//     Term 1 (APS4322-7000)/APS Outputs/Current D 1X0 <-> Data Pointer/DCurrentSetPoints[6]
//     Term 1 (APS4322-7000)/APS Outputs/Current D 1X1 <-> Data Pointer/DCurrentSetPoints[7]
//     Term 1 (APS4322-7000)/APS Outputs/Current D 1X2 <-> Data Pointer/DCurrentSetPoints[8]
//     Term 1 (APS4322-7000)/APS Outputs/Current D 2X0 <-> Data Pointer/DCurrentSetPoints[12]
//     Term 1 (APS4322-7000)/APS Outputs/Current D 2X1 <-> Data Pointer/DCurrentSetPoints[13]
//     Term 1 (APS4322-7000)/APS Outputs/Current D 2X2 <-> Data Pointer/DCurrentSetPoints[14]
//     Term 1 (APS4322-7000)/APS Outputs/Current D 3X0 <-> Data Pointer/DCurrentSetPoints[18]
//     Term 1 (APS4322-7000)/APS Outputs/Current D 3X1 <-> Data Pointer/DCurrentSetPoints[19]
//     Term 1 (APS4322-7000)/APS Outputs/Current D 3X2 <-> Data Pointer/DCurrentSetPoints[20]
//     Term 1 (APS4322-7000)/APS Outputs/Current D 0Y0 <-> Data Pointer/DCurrentSetPoints[3]
//     Term 1 (APS4322-7000)/APS Outputs/Current D 0Y1 <-> Data Pointer/DCurrentSetPoints[4]
//     Term 1 (APS4322-7000)/APS Outputs/Current D 0Y2 <-> Data Pointer/DCurrentSetPoints[5]
//     Term 1 (APS4322-7000)/APS Outputs/Current D 1Y0 <-> Data Pointer/DCurrentSetPoints[9]
//     Term 1 (APS4322-7000)/APS Outputs/Current D 1Y1 <-> Data Pointer/DCurrentSetPoints[10]
//     Term 1 (APS4322-7000)/APS Outputs/Current D 1Y2 <-> Data Pointer/DCurrentSetPoints[11]
//     Term 1 (APS4322-7000)/APS Outputs/Current D 2Y0 <-> Data Pointer/DCurrentSetPoints[15]
//     Term 1 (APS4322-7000)/APS Outputs/Current D 2Y1 <-> Data Pointer/DCurrentSetPoints[16]
//     Term 1 (APS4322-7000)/APS Outputs/Current D 2Y2 <-> Data Pointer/DCurrentSetPoints[17]
//     Term 1 (APS4322-7000)/APS Outputs/Current D 3Y0 <-> Data Pointer/DCurrentSetPoints[21]
//     Term 1 (APS4322-7000)/APS Outputs/Current D 3Y1 <-> Data Pointer/DCurrentSetPoints[22]
//     Term 1 (APS4322-7000)/APS Outputs/Current D 3Y2 <-> Data Pointer/DCurrentSetPoints[23]
//     Term 1 (APS4322-7000)/APS Outputs/Current Q 0X0 <-> Data Pointer/QCurrentSetPoints[0]
//     Term 1 (APS4322-7000)/APS Outputs/Current Q 0X1 <-> Data Pointer/QCurrentSetPoints[1]
//     Term 1 (APS4322-7000)/APS Outputs/Current Q 0X2 <-> Data Pointer/QCurrentSetPoints[2]
//     Term 1 (APS4322-7000)/APS Outputs/Current Q 1X0 <-> Data Pointer/QCurrentSetPoints[6]
//     Term 1 (APS4322-7000)/APS Outputs/Current Q 1X1 <-> Data Pointer/QCurrentSetPoints[7]
//     Term 1 (APS4322-7000)/APS Outputs/Current Q 1X2 <-> Data Pointer/QCurrentSetPoints[8]
//     Term 1 (APS4322-7000)/APS Outputs/Current Q 2X0 <-> Data Pointer/QCurrentSetPoints[12]
//     Term 1 (APS4322-7000)/APS Outputs/Current Q 2X1 <-> Data Pointer/QCurrentSetPoints[13]
//     Term 1 (APS4322-7000)/APS Outputs/Current Q 2X2 <-> Data Pointer/QCurrentSetPoints[14]
//     Term 1 (APS4322-7000)/APS Outputs/Current Q 3X0 <-> Data Pointer/QCurrentSetPoints[18]
//     Term 1 (APS4322-7000)/APS Outputs/Current Q 3X1 <-> Data Pointer/QCurrentSetPoints[19]
//     Term 1 (APS4322-7000)/APS Outputs/Current Q 3X2 <-> Data Pointer/QCurrentSetPoints[20]
//     Term 1 (APS4322-7000)/APS Outputs/Current Q 0Y0 <-> Data Pointer/QCurrentSetPoints[3]
//     Term 1 (APS4322-7000)/APS Outputs/Current Q 0Y1 <-> Data Pointer/QCurrentSetPoints[4]
//     Term 1 (APS4322-7000)/APS Outputs/Current Q 0Y2 <-> Data Pointer/QCurrentSetPoints[5]
//     Term 1 (APS4322-7000)/APS Outputs/Current Q 1Y0 <-> Data Pointer/QCurrentSetPoints[9]
//     Term 1 (APS4322-7000)/APS Outputs/Current Q 1Y1 <-> Data Pointer/QCurrentSetPoints[10]
//     Term 1 (APS4322-7000)/APS Outputs/Current Q 1Y2 <-> Data Pointer/QCurrentSetPoints[11]
//     Term 1 (APS4322-7000)/APS Outputs/Current Q 2Y0 <-> Data Pointer/QCurrentSetPoints[15]
//     Term 1 (APS4322-7000)/APS Outputs/Current Q 2Y1 <-> Data Pointer/QCurrentSetPoints[16]
//     Term 1 (APS4322-7000)/APS Outputs/Current Q 2Y2 <-> Data Pointer/QCurrentSetPoints[17]
//     Term 1 (APS4322-7000)/APS Outputs/Current Q 3Y0 <-> Data Pointer/QCurrentSetPoints[21]
//     Term 1 (APS4322-7000)/APS Outputs/Current Q 3Y1 <-> Data Pointer/QCurrentSetPoints[22]
//     Term 1 (APS4322-7000)/APS Outputs/Current Q 3Y2 <-> Data Pointer/QCurrentSetPoints[23]
//     Term 1 (APS4322-7000)/APS Outputs/PhiE 0X0 <-> Data Pointer/PhiSetPoints[0]
//     Term 1 (APS4322-7000)/APS Outputs/PhiE 0X1 <-> Data Pointer/PhiSetPoints[1]
//     Term 1 (APS4322-7000)/APS Outputs/PhiE 0X2 <-> Data Pointer/PhiSetPoints[2]
//     Term 1 (APS4322-7000)/APS Outputs/PhiE 1X0 <-> Data Pointer/PhiSetPoints[6]
//     Term 1 (APS4322-7000)/APS Outputs/PhiE 1X1 <-> Data Pointer/PhiSetPoints[7]
//     Term 1 (APS4322-7000)/APS Outputs/PhiE 1X2 <-> Data Pointer/PhiSetPoints[8]
//     Term 1 (APS4322-7000)/APS Outputs/PhiE 2X0 <-> Data Pointer/PhiSetPoints[12]
//     Term 1 (APS4322-7000)/APS Outputs/PhiE 2X1 <-> Data Pointer/PhiSetPoints[13]
//     Term 1 (APS4322-7000)/APS Outputs/PhiE 2X2 <-> Data Pointer/PhiSetPoints[14]
//     Term 1 (APS4322-7000)/APS Outputs/PhiE 3X0 <-> Data Pointer/PhiSetPoints[18]
//     Term 1 (APS4322-7000)/APS Outputs/PhiE 3X1 <-> Data Pointer/PhiSetPoints[19]
//     Term 1 (APS4322-7000)/APS Outputs/PhiE 3X2 <-> Data Pointer/PhiSetPoints[20]
//     Term 1 (APS4322-7000)/APS Outputs/PhiE 0Y0 <-> Data Pointer/PhiSetPoints[3]
//     Term 1 (APS4322-7000)/APS Outputs/PhiE 0Y1 <-> Data Pointer/PhiSetPoints[4]
//     Term 1 (APS4322-7000)/APS Outputs/PhiE 0Y2 <-> Data Pointer/PhiSetPoints[5]
//     Term 1 (APS4322-7000)/APS Outputs/PhiE 1Y0 <-> Data Pointer/PhiSetPoints[9]
//     Term 1 (APS4322-7000)/APS Outputs/PhiE 1Y1 <-> Data Pointer/PhiSetPoints[10]
//     Term 1 (APS4322-7000)/APS Outputs/PhiE 1Y2 <-> Data Pointer/PhiSetPoints[11]
//     Term 1 (APS4322-7000)/APS Outputs/PhiE 2Y0 <-> Data Pointer/PhiSetPoints[15]
//     Term 1 (APS4322-7000)/APS Outputs/PhiE 2Y1 <-> Data Pointer/PhiSetPoints[16]
//     Term 1 (APS4322-7000)/APS Outputs/PhiE 2Y2 <-> Data Pointer/PhiSetPoints[17]
//     Term 1 (APS4322-7000)/APS Outputs/PhiE 3Y0 <-> Data Pointer/PhiSetPoints[21]
//     Term 1 (APS4322-7000)/APS Outputs/PhiE 3Y1 <-> Data Pointer/PhiSetPoints[22]
//     Term 1 (APS4322-7000)/APS Outputs/PhiE 3Y2 <-> Data Pointer/PhiSetPoints[23]
//     Term 1 (APS4322-7000)/Term 2 (APS4322-5000)/FB Inputs/A{0..8 step 2} X-Field <-> Data Pointer/HallSensorFieldsXYZ[{0..12 step 3}]  (5 links)
//     Term 1 (APS4322-7000)/Term 2 (APS4322-5000)/FB Inputs/A{0..8 step 2} Y-Field <-> Data Pointer/HallSensorFieldsXYZ[{1..13 step 3}]  (5 links)
//     Term 1 (APS4322-7000)/Term 2 (APS4322-5000)/FB Inputs/A{0..8 step 2} Z-Field <-> Data Pointer/HallSensorFieldsXYZ[{2..14 step 3}]  (5 links)
//     Term 1 (APS4322-7000)/Term 2 (APS4322-5000)/FB Inputs/B{1..9 step 2} X-Field <-> Data Pointer/HallSensorFieldsXYZ[{15..27 step 3}]  (5 links)
//     Term 1 (APS4322-7000)/Term 2 (APS4322-5000)/FB Inputs/B{1..9 step 2} Y-Field <-> Data Pointer/HallSensorFieldsXYZ[{16..28 step 3}]  (5 links)
//     Term 1 (APS4322-7000)/Term 2 (APS4322-5000)/FB Inputs/B{1..9 step 2} Z-Field <-> Data Pointer/HallSensorFieldsXYZ[{17..29 step 3}]  (5 links)
//     Term 1 (APS4322-7000)/Term 2 (APS4322-5000)/FB Inputs/C{0..8 step 2} X-Field <-> Data Pointer/HallSensorFieldsXYZ[{30..42 step 3}]  (5 links)
//     Term 1 (APS4322-7000)/Term 2 (APS4322-5000)/FB Inputs/C{0..8 step 2} Y-Field <-> Data Pointer/HallSensorFieldsXYZ[{31..43 step 3}]  (5 links)
//     Term 1 (APS4322-7000)/Term 2 (APS4322-5000)/FB Inputs/C{0..8 step 2} Z-Field <-> Data Pointer/HallSensorFieldsXYZ[{32..44 step 3}]  (5 links)
//     Term 1 (APS4322-7000)/Term 2 (APS4322-5000)/FB Inputs/D{1..9 step 2} X-Field <-> Data Pointer/HallSensorFieldsXYZ[{45..57 step 3}]  (5 links)
//     Term 1 (APS4322-7000)/Term 2 (APS4322-5000)/FB Inputs/D{1..9 step 2} Y-Field <-> Data Pointer/HallSensorFieldsXYZ[{46..58 step 3}]  (5 links)
//     Term 1 (APS4322-7000)/Term 2 (APS4322-5000)/FB Inputs/D{1..9 step 2} Z-Field <-> Data Pointer/HallSensorFieldsXYZ[{47..59 step 3}]  (5 links)
//     Term 1 (APS4322-7000)/Term 2 (APS4322-5000)/FB Inputs/E{0..8 step 2} X-Field <-> Data Pointer/HallSensorFieldsXYZ[{60..72 step 3}]  (5 links)
//     Term 1 (APS4322-7000)/Term 2 (APS4322-5000)/FB Inputs/E{0..8 step 2} Y-Field <-> Data Pointer/HallSensorFieldsXYZ[{61..73 step 3}]  (5 links)
//     Term 1 (APS4322-7000)/Term 2 (APS4322-5000)/FB Inputs/E{0..8 step 2} Z-Field <-> Data Pointer/HallSensorFieldsXYZ[{62..74 step 3}]  (5 links)
//     Term 1 (APS4322-7000)/Term 2 (APS4322-5000)/FB Inputs/F{1..9 step 2} X-Field <-> Data Pointer/HallSensorFieldsXYZ[{75..87 step 3}]  (5 links)
//     Term 1 (APS4322-7000)/Term 2 (APS4322-5000)/FB Inputs/F{1..9 step 2} Y-Field <-> Data Pointer/HallSensorFieldsXYZ[{76..88 step 3}]  (5 links)
//     Term 1 (APS4322-7000)/Term 2 (APS4322-5000)/FB Inputs/F{1..9 step 2} Z-Field <-> Data Pointer/HallSensorFieldsXYZ[{77..89 step 3}]  (5 links)
//     Term 1 (APS4322-7000)/Term 2 (APS4322-5000)/FB Inputs/G{0..8 step 2} X-Field <-> Data Pointer/HallSensorFieldsXYZ[{90..102 step 3}]  (5 links)
//     Term 1 (APS4322-7000)/Term 2 (APS4322-5000)/FB Inputs/G{0..8 step 2} Y-Field <-> Data Pointer/HallSensorFieldsXYZ[{91..103 step 3}]  (5 links)
//     Term 1 (APS4322-7000)/Term 2 (APS4322-5000)/FB Inputs/G{0..8 step 2} Z-Field <-> Data Pointer/HallSensorFieldsXYZ[{92..104 step 3}]  (5 links)
//     Term 1 (APS4322-7000)/Term 2 (APS4322-5000)/FB Inputs/H{1..9 step 2} X-Field <-> Data Pointer/HallSensorFieldsXYZ[{105..117 step 3}]  (5 links)
//     Term 1 (APS4322-7000)/Term 2 (APS4322-5000)/FB Inputs/H{1..9 step 2} Y-Field <-> Data Pointer/HallSensorFieldsXYZ[{106..118 step 3}]  (5 links)
//     Term 1 (APS4322-7000)/Term 2 (APS4322-5000)/FB Inputs/H{1..9 step 2} Z-Field <-> Data Pointer/HallSensorFieldsXYZ[{107..119 step 3}]  (5 links)
//     Term 1 (APS4322-7000)/Term 2 (APS4322-5000)/FB Inputs/I{0..8 step 2} X-Field <-> Data Pointer/HallSensorFieldsXYZ[{120..132 step 3}]  (5 links)
//     Term 1 (APS4322-7000)/Term 2 (APS4322-5000)/FB Inputs/I{0..8 step 2} Y-Field <-> Data Pointer/HallSensorFieldsXYZ[{121..133 step 3}]  (5 links)
//     Term 1 (APS4322-7000)/Term 2 (APS4322-5000)/FB Inputs/I{0..8 step 2} Z-Field <-> Data Pointer/HallSensorFieldsXYZ[{122..134 step 3}]  (5 links)
//     Term 1 (APS4322-7000)/Term 2 (APS4322-5000)/FB Inputs/J{1..9 step 2} X-Field <-> Data Pointer/HallSensorFieldsXYZ[{135..147 step 3}]  (5 links)
//     Term 1 (APS4322-7000)/Term 2 (APS4322-5000)/FB Inputs/J{1..9 step 2} Y-Field <-> Data Pointer/HallSensorFieldsXYZ[{136..148 step 3}]  (5 links)
//     Term 1 (APS4322-7000)/Term 2 (APS4322-5000)/FB Inputs/J{1..9 step 2} Z-Field <-> Data Pointer/HallSensorFieldsXYZ[{137..149 step 3}]  (5 links)
//     Term 1 (APS4322-7000)/Term 2 (APS4322-5000)/FB Inputs/Status <-> Data Pointer/FeedbackStatus
//   Device 6 (EtherCAT) <-> TcCOM Objects/XPlanar/Part1/APS4322_P1_4
//     Term 3 (APS4322-7000)/APS Comm Inputs/CommStatusWord <-> Data Pointer/MoverCommStatusWord
//     Term 3 (APS4322-7000)/APS Comm Inputs/Data {1..4} <-> Data Pointer/MoverCommDataIn[{0..3}]  (4 links)
//     Term 3 (APS4322-7000)/APS Comm Outputs/CommControlWord <-> Data Pointer/MoverCommControlWord
//     Term 3 (APS4322-7000)/APS Comm Outputs/Data 1 <-> Data Pointer/MoverCommDataOut
//     Term 3 (APS4322-7000)/APS Diagdata/DC Link Voltage <-> Data Pointer/DcLinkVoltage
//     Term 3 (APS4322-7000)/APS Diagdata/Power supply current <-> Data Pointer/PowerSupplyCurrent
//     Term 3 (APS4322-7000)/APS Inputs/StatusWord <-> Data Pointer/PowerUnitStatusWord
//     Term 3 (APS4322-7000)/APS Outputs/ControlWord <-> Data Pointer/PowerUnitControlWord
//     Term 3 (APS4322-7000)/APS Outputs/Current D 0X0 <-> Data Pointer/DCurrentSetPoints[0]
//     Term 3 (APS4322-7000)/APS Outputs/Current D 0X1 <-> Data Pointer/DCurrentSetPoints[1]
//     Term 3 (APS4322-7000)/APS Outputs/Current D 0X2 <-> Data Pointer/DCurrentSetPoints[2]
//     Term 3 (APS4322-7000)/APS Outputs/Current D 1X0 <-> Data Pointer/DCurrentSetPoints[6]
//     Term 3 (APS4322-7000)/APS Outputs/Current D 1X1 <-> Data Pointer/DCurrentSetPoints[7]
//     Term 3 (APS4322-7000)/APS Outputs/Current D 1X2 <-> Data Pointer/DCurrentSetPoints[8]
//     Term 3 (APS4322-7000)/APS Outputs/Current D 2X0 <-> Data Pointer/DCurrentSetPoints[12]
//     Term 3 (APS4322-7000)/APS Outputs/Current D 2X1 <-> Data Pointer/DCurrentSetPoints[13]
//     Term 3 (APS4322-7000)/APS Outputs/Current D 2X2 <-> Data Pointer/DCurrentSetPoints[14]
//     Term 3 (APS4322-7000)/APS Outputs/Current D 3X0 <-> Data Pointer/DCurrentSetPoints[18]
//     Term 3 (APS4322-7000)/APS Outputs/Current D 3X1 <-> Data Pointer/DCurrentSetPoints[19]
//     Term 3 (APS4322-7000)/APS Outputs/Current D 3X2 <-> Data Pointer/DCurrentSetPoints[20]
//     Term 3 (APS4322-7000)/APS Outputs/Current D 0Y0 <-> Data Pointer/DCurrentSetPoints[3]
//     Term 3 (APS4322-7000)/APS Outputs/Current D 0Y1 <-> Data Pointer/DCurrentSetPoints[4]
//     Term 3 (APS4322-7000)/APS Outputs/Current D 0Y2 <-> Data Pointer/DCurrentSetPoints[5]
//     Term 3 (APS4322-7000)/APS Outputs/Current D 1Y0 <-> Data Pointer/DCurrentSetPoints[9]
//     Term 3 (APS4322-7000)/APS Outputs/Current D 1Y1 <-> Data Pointer/DCurrentSetPoints[10]
//     Term 3 (APS4322-7000)/APS Outputs/Current D 1Y2 <-> Data Pointer/DCurrentSetPoints[11]
//     Term 3 (APS4322-7000)/APS Outputs/Current D 2Y0 <-> Data Pointer/DCurrentSetPoints[15]
//     Term 3 (APS4322-7000)/APS Outputs/Current D 2Y1 <-> Data Pointer/DCurrentSetPoints[16]
//     Term 3 (APS4322-7000)/APS Outputs/Current D 2Y2 <-> Data Pointer/DCurrentSetPoints[17]
//     Term 3 (APS4322-7000)/APS Outputs/Current D 3Y0 <-> Data Pointer/DCurrentSetPoints[21]
//     Term 3 (APS4322-7000)/APS Outputs/Current D 3Y1 <-> Data Pointer/DCurrentSetPoints[22]
//     Term 3 (APS4322-7000)/APS Outputs/Current D 3Y2 <-> Data Pointer/DCurrentSetPoints[23]
//     Term 3 (APS4322-7000)/APS Outputs/Current Q 0X0 <-> Data Pointer/QCurrentSetPoints[0]
//     Term 3 (APS4322-7000)/APS Outputs/Current Q 0X1 <-> Data Pointer/QCurrentSetPoints[1]
//     Term 3 (APS4322-7000)/APS Outputs/Current Q 0X2 <-> Data Pointer/QCurrentSetPoints[2]
//     Term 3 (APS4322-7000)/APS Outputs/Current Q 1X0 <-> Data Pointer/QCurrentSetPoints[6]
//     Term 3 (APS4322-7000)/APS Outputs/Current Q 1X1 <-> Data Pointer/QCurrentSetPoints[7]
//     Term 3 (APS4322-7000)/APS Outputs/Current Q 1X2 <-> Data Pointer/QCurrentSetPoints[8]
//     Term 3 (APS4322-7000)/APS Outputs/Current Q 2X0 <-> Data Pointer/QCurrentSetPoints[12]
//     Term 3 (APS4322-7000)/APS Outputs/Current Q 2X1 <-> Data Pointer/QCurrentSetPoints[13]
//     Term 3 (APS4322-7000)/APS Outputs/Current Q 2X2 <-> Data Pointer/QCurrentSetPoints[14]
//     Term 3 (APS4322-7000)/APS Outputs/Current Q 3X0 <-> Data Pointer/QCurrentSetPoints[18]
//     Term 3 (APS4322-7000)/APS Outputs/Current Q 3X1 <-> Data Pointer/QCurrentSetPoints[19]
//     Term 3 (APS4322-7000)/APS Outputs/Current Q 3X2 <-> Data Pointer/QCurrentSetPoints[20]
//     Term 3 (APS4322-7000)/APS Outputs/Current Q 0Y0 <-> Data Pointer/QCurrentSetPoints[3]
//     Term 3 (APS4322-7000)/APS Outputs/Current Q 0Y1 <-> Data Pointer/QCurrentSetPoints[4]
//     Term 3 (APS4322-7000)/APS Outputs/Current Q 0Y2 <-> Data Pointer/QCurrentSetPoints[5]
//     Term 3 (APS4322-7000)/APS Outputs/Current Q 1Y0 <-> Data Pointer/QCurrentSetPoints[9]
//     Term 3 (APS4322-7000)/APS Outputs/Current Q 1Y1 <-> Data Pointer/QCurrentSetPoints[10]
//     Term 3 (APS4322-7000)/APS Outputs/Current Q 1Y2 <-> Data Pointer/QCurrentSetPoints[11]
//     Term 3 (APS4322-7000)/APS Outputs/Current Q 2Y0 <-> Data Pointer/QCurrentSetPoints[15]
//     Term 3 (APS4322-7000)/APS Outputs/Current Q 2Y1 <-> Data Pointer/QCurrentSetPoints[16]
//     Term 3 (APS4322-7000)/APS Outputs/Current Q 2Y2 <-> Data Pointer/QCurrentSetPoints[17]
//     Term 3 (APS4322-7000)/APS Outputs/Current Q 3Y0 <-> Data Pointer/QCurrentSetPoints[21]
//     Term 3 (APS4322-7000)/APS Outputs/Current Q 3Y1 <-> Data Pointer/QCurrentSetPoints[22]
//     Term 3 (APS4322-7000)/APS Outputs/Current Q 3Y2 <-> Data Pointer/QCurrentSetPoints[23]
//     Term 3 (APS4322-7000)/APS Outputs/PhiE 0X0 <-> Data Pointer/PhiSetPoints[0]
//     Term 3 (APS4322-7000)/APS Outputs/PhiE 0X1 <-> Data Pointer/PhiSetPoints[1]
//     Term 3 (APS4322-7000)/APS Outputs/PhiE 0X2 <-> Data Pointer/PhiSetPoints[2]
//     Term 3 (APS4322-7000)/APS Outputs/PhiE 1X0 <-> Data Pointer/PhiSetPoints[6]
//     Term 3 (APS4322-7000)/APS Outputs/PhiE 1X1 <-> Data Pointer/PhiSetPoints[7]
//     Term 3 (APS4322-7000)/APS Outputs/PhiE 1X2 <-> Data Pointer/PhiSetPoints[8]
//     Term 3 (APS4322-7000)/APS Outputs/PhiE 2X0 <-> Data Pointer/PhiSetPoints[12]
//     Term 3 (APS4322-7000)/APS Outputs/PhiE 2X1 <-> Data Pointer/PhiSetPoints[13]
//     Term 3 (APS4322-7000)/APS Outputs/PhiE 2X2 <-> Data Pointer/PhiSetPoints[14]
//     Term 3 (APS4322-7000)/APS Outputs/PhiE 3X0 <-> Data Pointer/PhiSetPoints[18]
//     Term 3 (APS4322-7000)/APS Outputs/PhiE 3X1 <-> Data Pointer/PhiSetPoints[19]
//     Term 3 (APS4322-7000)/APS Outputs/PhiE 3X2 <-> Data Pointer/PhiSetPoints[20]
//     Term 3 (APS4322-7000)/APS Outputs/PhiE 0Y0 <-> Data Pointer/PhiSetPoints[3]
//     Term 3 (APS4322-7000)/APS Outputs/PhiE 0Y1 <-> Data Pointer/PhiSetPoints[4]
//     Term 3 (APS4322-7000)/APS Outputs/PhiE 0Y2 <-> Data Pointer/PhiSetPoints[5]
//     Term 3 (APS4322-7000)/APS Outputs/PhiE 1Y0 <-> Data Pointer/PhiSetPoints[9]
//     Term 3 (APS4322-7000)/APS Outputs/PhiE 1Y1 <-> Data Pointer/PhiSetPoints[10]
//     Term 3 (APS4322-7000)/APS Outputs/PhiE 1Y2 <-> Data Pointer/PhiSetPoints[11]
//     Term 3 (APS4322-7000)/APS Outputs/PhiE 2Y0 <-> Data Pointer/PhiSetPoints[15]
//     Term 3 (APS4322-7000)/APS Outputs/PhiE 2Y1 <-> Data Pointer/PhiSetPoints[16]
//     Term 3 (APS4322-7000)/APS Outputs/PhiE 2Y2 <-> Data Pointer/PhiSetPoints[17]
//     Term 3 (APS4322-7000)/APS Outputs/PhiE 3Y0 <-> Data Pointer/PhiSetPoints[21]
//     Term 3 (APS4322-7000)/APS Outputs/PhiE 3Y1 <-> Data Pointer/PhiSetPoints[22]
//     Term 3 (APS4322-7000)/APS Outputs/PhiE 3Y2 <-> Data Pointer/PhiSetPoints[23]
//     Term 3 (APS4322-7000)/Term 4 (APS4322-5000)/FB Inputs/A{0..8 step 2} X-Field <-> Data Pointer/HallSensorFieldsXYZ[{0..12 step 3}]  (5 links)
//     Term 3 (APS4322-7000)/Term 4 (APS4322-5000)/FB Inputs/A{0..8 step 2} Y-Field <-> Data Pointer/HallSensorFieldsXYZ[{1..13 step 3}]  (5 links)
//     Term 3 (APS4322-7000)/Term 4 (APS4322-5000)/FB Inputs/A{0..8 step 2} Z-Field <-> Data Pointer/HallSensorFieldsXYZ[{2..14 step 3}]  (5 links)
//     Term 3 (APS4322-7000)/Term 4 (APS4322-5000)/FB Inputs/B{1..9 step 2} X-Field <-> Data Pointer/HallSensorFieldsXYZ[{15..27 step 3}]  (5 links)
//     Term 3 (APS4322-7000)/Term 4 (APS4322-5000)/FB Inputs/B{1..9 step 2} Y-Field <-> Data Pointer/HallSensorFieldsXYZ[{16..28 step 3}]  (5 links)
//     Term 3 (APS4322-7000)/Term 4 (APS4322-5000)/FB Inputs/B{1..9 step 2} Z-Field <-> Data Pointer/HallSensorFieldsXYZ[{17..29 step 3}]  (5 links)
//     Term 3 (APS4322-7000)/Term 4 (APS4322-5000)/FB Inputs/C{0..8 step 2} X-Field <-> Data Pointer/HallSensorFieldsXYZ[{30..42 step 3}]  (5 links)
//     Term 3 (APS4322-7000)/Term 4 (APS4322-5000)/FB Inputs/C{0..8 step 2} Y-Field <-> Data Pointer/HallSensorFieldsXYZ[{31..43 step 3}]  (5 links)
//     Term 3 (APS4322-7000)/Term 4 (APS4322-5000)/FB Inputs/C{0..8 step 2} Z-Field <-> Data Pointer/HallSensorFieldsXYZ[{32..44 step 3}]  (5 links)
//     Term 3 (APS4322-7000)/Term 4 (APS4322-5000)/FB Inputs/D{1..9 step 2} X-Field <-> Data Pointer/HallSensorFieldsXYZ[{45..57 step 3}]  (5 links)
//     Term 3 (APS4322-7000)/Term 4 (APS4322-5000)/FB Inputs/D{1..9 step 2} Y-Field <-> Data Pointer/HallSensorFieldsXYZ[{46..58 step 3}]  (5 links)
//     Term 3 (APS4322-7000)/Term 4 (APS4322-5000)/FB Inputs/D{1..9 step 2} Z-Field <-> Data Pointer/HallSensorFieldsXYZ[{47..59 step 3}]  (5 links)
//     Term 3 (APS4322-7000)/Term 4 (APS4322-5000)/FB Inputs/E{0..8 step 2} X-Field <-> Data Pointer/HallSensorFieldsXYZ[{60..72 step 3}]  (5 links)
//     Term 3 (APS4322-7000)/Term 4 (APS4322-5000)/FB Inputs/E{0..8 step 2} Y-Field <-> Data Pointer/HallSensorFieldsXYZ[{61..73 step 3}]  (5 links)
//     Term 3 (APS4322-7000)/Term 4 (APS4322-5000)/FB Inputs/E{0..8 step 2} Z-Field <-> Data Pointer/HallSensorFieldsXYZ[{62..74 step 3}]  (5 links)
//     Term 3 (APS4322-7000)/Term 4 (APS4322-5000)/FB Inputs/F{1..9 step 2} X-Field <-> Data Pointer/HallSensorFieldsXYZ[{75..87 step 3}]  (5 links)
//     Term 3 (APS4322-7000)/Term 4 (APS4322-5000)/FB Inputs/F{1..9 step 2} Y-Field <-> Data Pointer/HallSensorFieldsXYZ[{76..88 step 3}]  (5 links)
//     Term 3 (APS4322-7000)/Term 4 (APS4322-5000)/FB Inputs/F{1..9 step 2} Z-Field <-> Data Pointer/HallSensorFieldsXYZ[{77..89 step 3}]  (5 links)
//     Term 3 (APS4322-7000)/Term 4 (APS4322-5000)/FB Inputs/G{0..8 step 2} X-Field <-> Data Pointer/HallSensorFieldsXYZ[{90..102 step 3}]  (5 links)
//     Term 3 (APS4322-7000)/Term 4 (APS4322-5000)/FB Inputs/G{0..8 step 2} Y-Field <-> Data Pointer/HallSensorFieldsXYZ[{91..103 step 3}]  (5 links)
//     Term 3 (APS4322-7000)/Term 4 (APS4322-5000)/FB Inputs/G{0..8 step 2} Z-Field <-> Data Pointer/HallSensorFieldsXYZ[{92..104 step 3}]  (5 links)
//     Term 3 (APS4322-7000)/Term 4 (APS4322-5000)/FB Inputs/H{1..9 step 2} X-Field <-> Data Pointer/HallSensorFieldsXYZ[{105..117 step 3}]  (5 links)
//     Term 3 (APS4322-7000)/Term 4 (APS4322-5000)/FB Inputs/H{1..9 step 2} Y-Field <-> Data Pointer/HallSensorFieldsXYZ[{106..118 step 3}]  (5 links)
//     Term 3 (APS4322-7000)/Term 4 (APS4322-5000)/FB Inputs/H{1..9 step 2} Z-Field <-> Data Pointer/HallSensorFieldsXYZ[{107..119 step 3}]  (5 links)
//     Term 3 (APS4322-7000)/Term 4 (APS4322-5000)/FB Inputs/I{0..8 step 2} X-Field <-> Data Pointer/HallSensorFieldsXYZ[{120..132 step 3}]  (5 links)
//     Term 3 (APS4322-7000)/Term 4 (APS4322-5000)/FB Inputs/I{0..8 step 2} Y-Field <-> Data Pointer/HallSensorFieldsXYZ[{121..133 step 3}]  (5 links)
//     Term 3 (APS4322-7000)/Term 4 (APS4322-5000)/FB Inputs/I{0..8 step 2} Z-Field <-> Data Pointer/HallSensorFieldsXYZ[{122..134 step 3}]  (5 links)
//     Term 3 (APS4322-7000)/Term 4 (APS4322-5000)/FB Inputs/J{1..9 step 2} X-Field <-> Data Pointer/HallSensorFieldsXYZ[{135..147 step 3}]  (5 links)
//     Term 3 (APS4322-7000)/Term 4 (APS4322-5000)/FB Inputs/J{1..9 step 2} Y-Field <-> Data Pointer/HallSensorFieldsXYZ[{136..148 step 3}]  (5 links)
//     Term 3 (APS4322-7000)/Term 4 (APS4322-5000)/FB Inputs/J{1..9 step 2} Z-Field <-> Data Pointer/HallSensorFieldsXYZ[{137..149 step 3}]  (5 links)
//     Term 3 (APS4322-7000)/Term 4 (APS4322-5000)/FB Inputs/Status <-> Data Pointer/FeedbackStatus
//   Device 6 (EtherCAT) <-> TcCOM Objects/XPlanar/Part1/APS4322_P1_7
//     Term 5 (APS4322-7000)/APS Comm Inputs/CommStatusWord <-> Data Pointer/MoverCommStatusWord
//     Term 5 (APS4322-7000)/APS Comm Inputs/Data {1..4} <-> Data Pointer/MoverCommDataIn[{0..3}]  (4 links)
//     Term 5 (APS4322-7000)/APS Comm Outputs/CommControlWord <-> Data Pointer/MoverCommControlWord
//     Term 5 (APS4322-7000)/APS Comm Outputs/Data 1 <-> Data Pointer/MoverCommDataOut
//     Term 5 (APS4322-7000)/APS Diagdata/DC Link Voltage <-> Data Pointer/DcLinkVoltage
//     Term 5 (APS4322-7000)/APS Diagdata/Power supply current <-> Data Pointer/PowerSupplyCurrent
//     Term 5 (APS4322-7000)/APS Inputs/StatusWord <-> Data Pointer/PowerUnitStatusWord
//     Term 5 (APS4322-7000)/APS Outputs/ControlWord <-> Data Pointer/PowerUnitControlWord
//     Term 5 (APS4322-7000)/APS Outputs/Current D 0X0 <-> Data Pointer/DCurrentSetPoints[0]
//     Term 5 (APS4322-7000)/APS Outputs/Current D 0X1 <-> Data Pointer/DCurrentSetPoints[1]
//     Term 5 (APS4322-7000)/APS Outputs/Current D 0X2 <-> Data Pointer/DCurrentSetPoints[2]
//     Term 5 (APS4322-7000)/APS Outputs/Current D 1X0 <-> Data Pointer/DCurrentSetPoints[6]
//     Term 5 (APS4322-7000)/APS Outputs/Current D 1X1 <-> Data Pointer/DCurrentSetPoints[7]
//     Term 5 (APS4322-7000)/APS Outputs/Current D 1X2 <-> Data Pointer/DCurrentSetPoints[8]
//     Term 5 (APS4322-7000)/APS Outputs/Current D 2X0 <-> Data Pointer/DCurrentSetPoints[12]
//     Term 5 (APS4322-7000)/APS Outputs/Current D 2X1 <-> Data Pointer/DCurrentSetPoints[13]
//     Term 5 (APS4322-7000)/APS Outputs/Current D 2X2 <-> Data Pointer/DCurrentSetPoints[14]
//     Term 5 (APS4322-7000)/APS Outputs/Current D 3X0 <-> Data Pointer/DCurrentSetPoints[18]
//     Term 5 (APS4322-7000)/APS Outputs/Current D 3X1 <-> Data Pointer/DCurrentSetPoints[19]
//     Term 5 (APS4322-7000)/APS Outputs/Current D 3X2 <-> Data Pointer/DCurrentSetPoints[20]
//     Term 5 (APS4322-7000)/APS Outputs/Current D 0Y0 <-> Data Pointer/DCurrentSetPoints[3]
//     Term 5 (APS4322-7000)/APS Outputs/Current D 0Y1 <-> Data Pointer/DCurrentSetPoints[4]
//     Term 5 (APS4322-7000)/APS Outputs/Current D 0Y2 <-> Data Pointer/DCurrentSetPoints[5]
//     Term 5 (APS4322-7000)/APS Outputs/Current D 1Y0 <-> Data Pointer/DCurrentSetPoints[9]
//     Term 5 (APS4322-7000)/APS Outputs/Current D 1Y1 <-> Data Pointer/DCurrentSetPoints[10]
//     Term 5 (APS4322-7000)/APS Outputs/Current D 1Y2 <-> Data Pointer/DCurrentSetPoints[11]
//     Term 5 (APS4322-7000)/APS Outputs/Current D 2Y0 <-> Data Pointer/DCurrentSetPoints[15]
//     Term 5 (APS4322-7000)/APS Outputs/Current D 2Y1 <-> Data Pointer/DCurrentSetPoints[16]
//     Term 5 (APS4322-7000)/APS Outputs/Current D 2Y2 <-> Data Pointer/DCurrentSetPoints[17]
//     Term 5 (APS4322-7000)/APS Outputs/Current D 3Y0 <-> Data Pointer/DCurrentSetPoints[21]
//     Term 5 (APS4322-7000)/APS Outputs/Current D 3Y1 <-> Data Pointer/DCurrentSetPoints[22]
//     Term 5 (APS4322-7000)/APS Outputs/Current D 3Y2 <-> Data Pointer/DCurrentSetPoints[23]
//     Term 5 (APS4322-7000)/APS Outputs/Current Q 0X0 <-> Data Pointer/QCurrentSetPoints[0]
//     Term 5 (APS4322-7000)/APS Outputs/Current Q 0X1 <-> Data Pointer/QCurrentSetPoints[1]
//     Term 5 (APS4322-7000)/APS Outputs/Current Q 0X2 <-> Data Pointer/QCurrentSetPoints[2]
//     Term 5 (APS4322-7000)/APS Outputs/Current Q 1X0 <-> Data Pointer/QCurrentSetPoints[6]
//     Term 5 (APS4322-7000)/APS Outputs/Current Q 1X1 <-> Data Pointer/QCurrentSetPoints[7]
//     Term 5 (APS4322-7000)/APS Outputs/Current Q 1X2 <-> Data Pointer/QCurrentSetPoints[8]
//     Term 5 (APS4322-7000)/APS Outputs/Current Q 2X0 <-> Data Pointer/QCurrentSetPoints[12]
//     Term 5 (APS4322-7000)/APS Outputs/Current Q 2X1 <-> Data Pointer/QCurrentSetPoints[13]
//     Term 5 (APS4322-7000)/APS Outputs/Current Q 2X2 <-> Data Pointer/QCurrentSetPoints[14]
//     Term 5 (APS4322-7000)/APS Outputs/Current Q 3X0 <-> Data Pointer/QCurrentSetPoints[18]
//     Term 5 (APS4322-7000)/APS Outputs/Current Q 3X1 <-> Data Pointer/QCurrentSetPoints[19]
//     Term 5 (APS4322-7000)/APS Outputs/Current Q 3X2 <-> Data Pointer/QCurrentSetPoints[20]
//     Term 5 (APS4322-7000)/APS Outputs/Current Q 0Y0 <-> Data Pointer/QCurrentSetPoints[3]
//     Term 5 (APS4322-7000)/APS Outputs/Current Q 0Y1 <-> Data Pointer/QCurrentSetPoints[4]
//     Term 5 (APS4322-7000)/APS Outputs/Current Q 0Y2 <-> Data Pointer/QCurrentSetPoints[5]
//     Term 5 (APS4322-7000)/APS Outputs/Current Q 1Y0 <-> Data Pointer/QCurrentSetPoints[9]
//     Term 5 (APS4322-7000)/APS Outputs/Current Q 1Y1 <-> Data Pointer/QCurrentSetPoints[10]
//     Term 5 (APS4322-7000)/APS Outputs/Current Q 1Y2 <-> Data Pointer/QCurrentSetPoints[11]
//     Term 5 (APS4322-7000)/APS Outputs/Current Q 2Y0 <-> Data Pointer/QCurrentSetPoints[15]
//     Term 5 (APS4322-7000)/APS Outputs/Current Q 2Y1 <-> Data Pointer/QCurrentSetPoints[16]
//     Term 5 (APS4322-7000)/APS Outputs/Current Q 2Y2 <-> Data Pointer/QCurrentSetPoints[17]
//     Term 5 (APS4322-7000)/APS Outputs/Current Q 3Y0 <-> Data Pointer/QCurrentSetPoints[21]
//     Term 5 (APS4322-7000)/APS Outputs/Current Q 3Y1 <-> Data Pointer/QCurrentSetPoints[22]
//     Term 5 (APS4322-7000)/APS Outputs/Current Q 3Y2 <-> Data Pointer/QCurrentSetPoints[23]
//     Term 5 (APS4322-7000)/APS Outputs/PhiE 0X0 <-> Data Pointer/PhiSetPoints[0]
//     Term 5 (APS4322-7000)/APS Outputs/PhiE 0X1 <-> Data Pointer/PhiSetPoints[1]
//     Term 5 (APS4322-7000)/APS Outputs/PhiE 0X2 <-> Data Pointer/PhiSetPoints[2]
//     Term 5 (APS4322-7000)/APS Outputs/PhiE 1X0 <-> Data Pointer/PhiSetPoints[6]
//     Term 5 (APS4322-7000)/APS Outputs/PhiE 1X1 <-> Data Pointer/PhiSetPoints[7]
//     Term 5 (APS4322-7000)/APS Outputs/PhiE 1X2 <-> Data Pointer/PhiSetPoints[8]
//     Term 5 (APS4322-7000)/APS Outputs/PhiE 2X0 <-> Data Pointer/PhiSetPoints[12]
//     Term 5 (APS4322-7000)/APS Outputs/PhiE 2X1 <-> Data Pointer/PhiSetPoints[13]
//     Term 5 (APS4322-7000)/APS Outputs/PhiE 2X2 <-> Data Pointer/PhiSetPoints[14]
//     Term 5 (APS4322-7000)/APS Outputs/PhiE 3X0 <-> Data Pointer/PhiSetPoints[18]
//     Term 5 (APS4322-7000)/APS Outputs/PhiE 3X1 <-> Data Pointer/PhiSetPoints[19]
//     Term 5 (APS4322-7000)/APS Outputs/PhiE 3X2 <-> Data Pointer/PhiSetPoints[20]
//     Term 5 (APS4322-7000)/APS Outputs/PhiE 0Y0 <-> Data Pointer/PhiSetPoints[3]
//     Term 5 (APS4322-7000)/APS Outputs/PhiE 0Y1 <-> Data Pointer/PhiSetPoints[4]
//     Term 5 (APS4322-7000)/APS Outputs/PhiE 0Y2 <-> Data Pointer/PhiSetPoints[5]
//     Term 5 (APS4322-7000)/APS Outputs/PhiE 1Y0 <-> Data Pointer/PhiSetPoints[9]
//     Term 5 (APS4322-7000)/APS Outputs/PhiE 1Y1 <-> Data Pointer/PhiSetPoints[10]
//     Term 5 (APS4322-7000)/APS Outputs/PhiE 1Y2 <-> Data Pointer/PhiSetPoints[11]
//     Term 5 (APS4322-7000)/APS Outputs/PhiE 2Y0 <-> Data Pointer/PhiSetPoints[15]
//     Term 5 (APS4322-7000)/APS Outputs/PhiE 2Y1 <-> Data Pointer/PhiSetPoints[16]
//     Term 5 (APS4322-7000)/APS Outputs/PhiE 2Y2 <-> Data Pointer/PhiSetPoints[17]
//     Term 5 (APS4322-7000)/APS Outputs/PhiE 3Y0 <-> Data Pointer/PhiSetPoints[21]
//     Term 5 (APS4322-7000)/APS Outputs/PhiE 3Y1 <-> Data Pointer/PhiSetPoints[22]
//     Term 5 (APS4322-7000)/APS Outputs/PhiE 3Y2 <-> Data Pointer/PhiSetPoints[23]
//     Term 5 (APS4322-7000)/Term 6 (APS4322-5000)/FB Inputs/A{0..8 step 2} X-Field <-> Data Pointer/HallSensorFieldsXYZ[{0..12 step 3}]  (5 links)
//     Term 5 (APS4322-7000)/Term 6 (APS4322-5000)/FB Inputs/A{0..8 step 2} Y-Field <-> Data Pointer/HallSensorFieldsXYZ[{1..13 step 3}]  (5 links)
//     Term 5 (APS4322-7000)/Term 6 (APS4322-5000)/FB Inputs/A{0..8 step 2} Z-Field <-> Data Pointer/HallSensorFieldsXYZ[{2..14 step 3}]  (5 links)
//     Term 5 (APS4322-7000)/Term 6 (APS4322-5000)/FB Inputs/B{1..9 step 2} X-Field <-> Data Pointer/HallSensorFieldsXYZ[{15..27 step 3}]  (5 links)
//     Term 5 (APS4322-7000)/Term 6 (APS4322-5000)/FB Inputs/B{1..9 step 2} Y-Field <-> Data Pointer/HallSensorFieldsXYZ[{16..28 step 3}]  (5 links)
//     Term 5 (APS4322-7000)/Term 6 (APS4322-5000)/FB Inputs/B{1..9 step 2} Z-Field <-> Data Pointer/HallSensorFieldsXYZ[{17..29 step 3}]  (5 links)
//     Term 5 (APS4322-7000)/Term 6 (APS4322-5000)/FB Inputs/C{0..8 step 2} X-Field <-> Data Pointer/HallSensorFieldsXYZ[{30..42 step 3}]  (5 links)
//     Term 5 (APS4322-7000)/Term 6 (APS4322-5000)/FB Inputs/C{0..8 step 2} Y-Field <-> Data Pointer/HallSensorFieldsXYZ[{31..43 step 3}]  (5 links)
//     Term 5 (APS4322-7000)/Term 6 (APS4322-5000)/FB Inputs/C{0..8 step 2} Z-Field <-> Data Pointer/HallSensorFieldsXYZ[{32..44 step 3}]  (5 links)
//     Term 5 (APS4322-7000)/Term 6 (APS4322-5000)/FB Inputs/D{1..9 step 2} X-Field <-> Data Pointer/HallSensorFieldsXYZ[{45..57 step 3}]  (5 links)
//     Term 5 (APS4322-7000)/Term 6 (APS4322-5000)/FB Inputs/D{1..9 step 2} Y-Field <-> Data Pointer/HallSensorFieldsXYZ[{46..58 step 3}]  (5 links)
//     Term 5 (APS4322-7000)/Term 6 (APS4322-5000)/FB Inputs/D{1..9 step 2} Z-Field <-> Data Pointer/HallSensorFieldsXYZ[{47..59 step 3}]  (5 links)
//     Term 5 (APS4322-7000)/Term 6 (APS4322-5000)/FB Inputs/E{0..8 step 2} X-Field <-> Data Pointer/HallSensorFieldsXYZ[{60..72 step 3}]  (5 links)
//     Term 5 (APS4322-7000)/Term 6 (APS4322-5000)/FB Inputs/E{0..8 step 2} Y-Field <-> Data Pointer/HallSensorFieldsXYZ[{61..73 step 3}]  (5 links)
//     Term 5 (APS4322-7000)/Term 6 (APS4322-5000)/FB Inputs/E{0..8 step 2} Z-Field <-> Data Pointer/HallSensorFieldsXYZ[{62..74 step 3}]  (5 links)
//     Term 5 (APS4322-7000)/Term 6 (APS4322-5000)/FB Inputs/F{1..9 step 2} X-Field <-> Data Pointer/HallSensorFieldsXYZ[{75..87 step 3}]  (5 links)
//     Term 5 (APS4322-7000)/Term 6 (APS4322-5000)/FB Inputs/F{1..9 step 2} Y-Field <-> Data Pointer/HallSensorFieldsXYZ[{76..88 step 3}]  (5 links)
//     Term 5 (APS4322-7000)/Term 6 (APS4322-5000)/FB Inputs/F{1..9 step 2} Z-Field <-> Data Pointer/HallSensorFieldsXYZ[{77..89 step 3}]  (5 links)
//     Term 5 (APS4322-7000)/Term 6 (APS4322-5000)/FB Inputs/G{0..8 step 2} X-Field <-> Data Pointer/HallSensorFieldsXYZ[{90..102 step 3}]  (5 links)
//     Term 5 (APS4322-7000)/Term 6 (APS4322-5000)/FB Inputs/G{0..8 step 2} Y-Field <-> Data Pointer/HallSensorFieldsXYZ[{91..103 step 3}]  (5 links)
//     Term 5 (APS4322-7000)/Term 6 (APS4322-5000)/FB Inputs/G{0..8 step 2} Z-Field <-> Data Pointer/HallSensorFieldsXYZ[{92..104 step 3}]  (5 links)
//     Term 5 (APS4322-7000)/Term 6 (APS4322-5000)/FB Inputs/H{1..9 step 2} X-Field <-> Data Pointer/HallSensorFieldsXYZ[{105..117 step 3}]  (5 links)
//     Term 5 (APS4322-7000)/Term 6 (APS4322-5000)/FB Inputs/H{1..9 step 2} Y-Field <-> Data Pointer/HallSensorFieldsXYZ[{106..118 step 3}]  (5 links)
//     Term 5 (APS4322-7000)/Term 6 (APS4322-5000)/FB Inputs/H{1..9 step 2} Z-Field <-> Data Pointer/HallSensorFieldsXYZ[{107..119 step 3}]  (5 links)
//     Term 5 (APS4322-7000)/Term 6 (APS4322-5000)/FB Inputs/I{0..8 step 2} X-Field <-> Data Pointer/HallSensorFieldsXYZ[{120..132 step 3}]  (5 links)
//     Term 5 (APS4322-7000)/Term 6 (APS4322-5000)/FB Inputs/I{0..8 step 2} Y-Field <-> Data Pointer/HallSensorFieldsXYZ[{121..133 step 3}]  (5 links)
//     Term 5 (APS4322-7000)/Term 6 (APS4322-5000)/FB Inputs/I{0..8 step 2} Z-Field <-> Data Pointer/HallSensorFieldsXYZ[{122..134 step 3}]  (5 links)
//     Term 5 (APS4322-7000)/Term 6 (APS4322-5000)/FB Inputs/J{1..9 step 2} X-Field <-> Data Pointer/HallSensorFieldsXYZ[{135..147 step 3}]  (5 links)
//     Term 5 (APS4322-7000)/Term 6 (APS4322-5000)/FB Inputs/J{1..9 step 2} Y-Field <-> Data Pointer/HallSensorFieldsXYZ[{136..148 step 3}]  (5 links)
//     Term 5 (APS4322-7000)/Term 6 (APS4322-5000)/FB Inputs/J{1..9 step 2} Z-Field <-> Data Pointer/HallSensorFieldsXYZ[{137..149 step 3}]  (5 links)
//     Term 5 (APS4322-7000)/Term 6 (APS4322-5000)/FB Inputs/Status <-> Data Pointer/FeedbackStatus
//   Device 6 (EtherCAT) <-> TcCOM Objects/XPlanar/Part1/APS4322_P1_8
//     Term 7 (APS4322-7000)/APS Comm Inputs/CommStatusWord <-> Data Pointer/MoverCommStatusWord
//     Term 7 (APS4322-7000)/APS Comm Inputs/Data {1..4} <-> Data Pointer/MoverCommDataIn[{0..3}]  (4 links)
//     Term 7 (APS4322-7000)/APS Comm Outputs/CommControlWord <-> Data Pointer/MoverCommControlWord
//     Term 7 (APS4322-7000)/APS Comm Outputs/Data 1 <-> Data Pointer/MoverCommDataOut
//     Term 7 (APS4322-7000)/APS Diagdata/DC Link Voltage <-> Data Pointer/DcLinkVoltage
//     Term 7 (APS4322-7000)/APS Diagdata/Power supply current <-> Data Pointer/PowerSupplyCurrent
//     Term 7 (APS4322-7000)/APS Inputs/StatusWord <-> Data Pointer/PowerUnitStatusWord
//     Term 7 (APS4322-7000)/APS Outputs/ControlWord <-> Data Pointer/PowerUnitControlWord
//     Term 7 (APS4322-7000)/APS Outputs/Current D 0X0 <-> Data Pointer/DCurrentSetPoints[0]
//     Term 7 (APS4322-7000)/APS Outputs/Current D 0X1 <-> Data Pointer/DCurrentSetPoints[1]
//     Term 7 (APS4322-7000)/APS Outputs/Current D 0X2 <-> Data Pointer/DCurrentSetPoints[2]
//     Term 7 (APS4322-7000)/APS Outputs/Current D 1X0 <-> Data Pointer/DCurrentSetPoints[6]
//     Term 7 (APS4322-7000)/APS Outputs/Current D 1X1 <-> Data Pointer/DCurrentSetPoints[7]
//     Term 7 (APS4322-7000)/APS Outputs/Current D 1X2 <-> Data Pointer/DCurrentSetPoints[8]
//     Term 7 (APS4322-7000)/APS Outputs/Current D 2X0 <-> Data Pointer/DCurrentSetPoints[12]
//     Term 7 (APS4322-7000)/APS Outputs/Current D 2X1 <-> Data Pointer/DCurrentSetPoints[13]
//     Term 7 (APS4322-7000)/APS Outputs/Current D 2X2 <-> Data Pointer/DCurrentSetPoints[14]
//     Term 7 (APS4322-7000)/APS Outputs/Current D 3X0 <-> Data Pointer/DCurrentSetPoints[18]
//     Term 7 (APS4322-7000)/APS Outputs/Current D 3X1 <-> Data Pointer/DCurrentSetPoints[19]
//     Term 7 (APS4322-7000)/APS Outputs/Current D 3X2 <-> Data Pointer/DCurrentSetPoints[20]
//     Term 7 (APS4322-7000)/APS Outputs/Current D 0Y0 <-> Data Pointer/DCurrentSetPoints[3]
//     Term 7 (APS4322-7000)/APS Outputs/Current D 0Y1 <-> Data Pointer/DCurrentSetPoints[4]
//     Term 7 (APS4322-7000)/APS Outputs/Current D 0Y2 <-> Data Pointer/DCurrentSetPoints[5]
//     Term 7 (APS4322-7000)/APS Outputs/Current D 1Y0 <-> Data Pointer/DCurrentSetPoints[9]
//     Term 7 (APS4322-7000)/APS Outputs/Current D 1Y1 <-> Data Pointer/DCurrentSetPoints[10]
//     Term 7 (APS4322-7000)/APS Outputs/Current D 1Y2 <-> Data Pointer/DCurrentSetPoints[11]
//     Term 7 (APS4322-7000)/APS Outputs/Current D 2Y0 <-> Data Pointer/DCurrentSetPoints[15]
//     Term 7 (APS4322-7000)/APS Outputs/Current D 2Y1 <-> Data Pointer/DCurrentSetPoints[16]
//     Term 7 (APS4322-7000)/APS Outputs/Current D 2Y2 <-> Data Pointer/DCurrentSetPoints[17]
//     Term 7 (APS4322-7000)/APS Outputs/Current D 3Y0 <-> Data Pointer/DCurrentSetPoints[21]
//     Term 7 (APS4322-7000)/APS Outputs/Current D 3Y1 <-> Data Pointer/DCurrentSetPoints[22]
//     Term 7 (APS4322-7000)/APS Outputs/Current D 3Y2 <-> Data Pointer/DCurrentSetPoints[23]
//     Term 7 (APS4322-7000)/APS Outputs/Current Q 0X0 <-> Data Pointer/QCurrentSetPoints[0]
//     Term 7 (APS4322-7000)/APS Outputs/Current Q 0X1 <-> Data Pointer/QCurrentSetPoints[1]
//     Term 7 (APS4322-7000)/APS Outputs/Current Q 0X2 <-> Data Pointer/QCurrentSetPoints[2]
//     Term 7 (APS4322-7000)/APS Outputs/Current Q 1X0 <-> Data Pointer/QCurrentSetPoints[6]
//     Term 7 (APS4322-7000)/APS Outputs/Current Q 1X1 <-> Data Pointer/QCurrentSetPoints[7]
//     Term 7 (APS4322-7000)/APS Outputs/Current Q 1X2 <-> Data Pointer/QCurrentSetPoints[8]
//     Term 7 (APS4322-7000)/APS Outputs/Current Q 2X0 <-> Data Pointer/QCurrentSetPoints[12]
//     Term 7 (APS4322-7000)/APS Outputs/Current Q 2X1 <-> Data Pointer/QCurrentSetPoints[13]
//     Term 7 (APS4322-7000)/APS Outputs/Current Q 2X2 <-> Data Pointer/QCurrentSetPoints[14]
//     Term 7 (APS4322-7000)/APS Outputs/Current Q 3X0 <-> Data Pointer/QCurrentSetPoints[18]
//     Term 7 (APS4322-7000)/APS Outputs/Current Q 3X1 <-> Data Pointer/QCurrentSetPoints[19]
//     Term 7 (APS4322-7000)/APS Outputs/Current Q 3X2 <-> Data Pointer/QCurrentSetPoints[20]
//     Term 7 (APS4322-7000)/APS Outputs/Current Q 0Y0 <-> Data Pointer/QCurrentSetPoints[3]
//     Term 7 (APS4322-7000)/APS Outputs/Current Q 0Y1 <-> Data Pointer/QCurrentSetPoints[4]
//     Term 7 (APS4322-7000)/APS Outputs/Current Q 0Y2 <-> Data Pointer/QCurrentSetPoints[5]
//     Term 7 (APS4322-7000)/APS Outputs/Current Q 1Y0 <-> Data Pointer/QCurrentSetPoints[9]
//     Term 7 (APS4322-7000)/APS Outputs/Current Q 1Y1 <-> Data Pointer/QCurrentSetPoints[10]
//     Term 7 (APS4322-7000)/APS Outputs/Current Q 1Y2 <-> Data Pointer/QCurrentSetPoints[11]
//     Term 7 (APS4322-7000)/APS Outputs/Current Q 2Y0 <-> Data Pointer/QCurrentSetPoints[15]
//     Term 7 (APS4322-7000)/APS Outputs/Current Q 2Y1 <-> Data Pointer/QCurrentSetPoints[16]
//     Term 7 (APS4322-7000)/APS Outputs/Current Q 2Y2 <-> Data Pointer/QCurrentSetPoints[17]
//     Term 7 (APS4322-7000)/APS Outputs/Current Q 3Y0 <-> Data Pointer/QCurrentSetPoints[21]
//     Term 7 (APS4322-7000)/APS Outputs/Current Q 3Y1 <-> Data Pointer/QCurrentSetPoints[22]
//     Term 7 (APS4322-7000)/APS Outputs/Current Q 3Y2 <-> Data Pointer/QCurrentSetPoints[23]
//     Term 7 (APS4322-7000)/APS Outputs/PhiE 0X0 <-> Data Pointer/PhiSetPoints[0]
//     Term 7 (APS4322-7000)/APS Outputs/PhiE 0X1 <-> Data Pointer/PhiSetPoints[1]
//     Term 7 (APS4322-7000)/APS Outputs/PhiE 0X2 <-> Data Pointer/PhiSetPoints[2]
//     Term 7 (APS4322-7000)/APS Outputs/PhiE 1X0 <-> Data Pointer/PhiSetPoints[6]
//     Term 7 (APS4322-7000)/APS Outputs/PhiE 1X1 <-> Data Pointer/PhiSetPoints[7]
//     Term 7 (APS4322-7000)/APS Outputs/PhiE 1X2 <-> Data Pointer/PhiSetPoints[8]
//     Term 7 (APS4322-7000)/APS Outputs/PhiE 2X0 <-> Data Pointer/PhiSetPoints[12]
//     Term 7 (APS4322-7000)/APS Outputs/PhiE 2X1 <-> Data Pointer/PhiSetPoints[13]
//     Term 7 (APS4322-7000)/APS Outputs/PhiE 2X2 <-> Data Pointer/PhiSetPoints[14]
//     Term 7 (APS4322-7000)/APS Outputs/PhiE 3X0 <-> Data Pointer/PhiSetPoints[18]
//     Term 7 (APS4322-7000)/APS Outputs/PhiE 3X1 <-> Data Pointer/PhiSetPoints[19]
//     Term 7 (APS4322-7000)/APS Outputs/PhiE 3X2 <-> Data Pointer/PhiSetPoints[20]
//     Term 7 (APS4322-7000)/APS Outputs/PhiE 0Y0 <-> Data Pointer/PhiSetPoints[3]
//     Term 7 (APS4322-7000)/APS Outputs/PhiE 0Y1 <-> Data Pointer/PhiSetPoints[4]
//     Term 7 (APS4322-7000)/APS Outputs/PhiE 0Y2 <-> Data Pointer/PhiSetPoints[5]
//     Term 7 (APS4322-7000)/APS Outputs/PhiE 1Y0 <-> Data Pointer/PhiSetPoints[9]
//     Term 7 (APS4322-7000)/APS Outputs/PhiE 1Y1 <-> Data Pointer/PhiSetPoints[10]
//     Term 7 (APS4322-7000)/APS Outputs/PhiE 1Y2 <-> Data Pointer/PhiSetPoints[11]
//     Term 7 (APS4322-7000)/APS Outputs/PhiE 2Y0 <-> Data Pointer/PhiSetPoints[15]
//     Term 7 (APS4322-7000)/APS Outputs/PhiE 2Y1 <-> Data Pointer/PhiSetPoints[16]
//     Term 7 (APS4322-7000)/APS Outputs/PhiE 2Y2 <-> Data Pointer/PhiSetPoints[17]
//     Term 7 (APS4322-7000)/APS Outputs/PhiE 3Y0 <-> Data Pointer/PhiSetPoints[21]
//     Term 7 (APS4322-7000)/APS Outputs/PhiE 3Y1 <-> Data Pointer/PhiSetPoints[22]
//     Term 7 (APS4322-7000)/APS Outputs/PhiE 3Y2 <-> Data Pointer/PhiSetPoints[23]
//     Term 7 (APS4322-7000)/Term 8 (APS4322-5000)/FB Inputs/A{0..8 step 2} X-Field <-> Data Pointer/HallSensorFieldsXYZ[{0..12 step 3}]  (5 links)
//     Term 7 (APS4322-7000)/Term 8 (APS4322-5000)/FB Inputs/A{0..8 step 2} Y-Field <-> Data Pointer/HallSensorFieldsXYZ[{1..13 step 3}]  (5 links)
//     Term 7 (APS4322-7000)/Term 8 (APS4322-5000)/FB Inputs/A{0..8 step 2} Z-Field <-> Data Pointer/HallSensorFieldsXYZ[{2..14 step 3}]  (5 links)
//     Term 7 (APS4322-7000)/Term 8 (APS4322-5000)/FB Inputs/B{1..9 step 2} X-Field <-> Data Pointer/HallSensorFieldsXYZ[{15..27 step 3}]  (5 links)
//     Term 7 (APS4322-7000)/Term 8 (APS4322-5000)/FB Inputs/B{1..9 step 2} Y-Field <-> Data Pointer/HallSensorFieldsXYZ[{16..28 step 3}]  (5 links)
//     Term 7 (APS4322-7000)/Term 8 (APS4322-5000)/FB Inputs/B{1..9 step 2} Z-Field <-> Data Pointer/HallSensorFieldsXYZ[{17..29 step 3}]  (5 links)
//     Term 7 (APS4322-7000)/Term 8 (APS4322-5000)/FB Inputs/C{0..8 step 2} X-Field <-> Data Pointer/HallSensorFieldsXYZ[{30..42 step 3}]  (5 links)
//     Term 7 (APS4322-7000)/Term 8 (APS4322-5000)/FB Inputs/C{0..8 step 2} Y-Field <-> Data Pointer/HallSensorFieldsXYZ[{31..43 step 3}]  (5 links)
//     Term 7 (APS4322-7000)/Term 8 (APS4322-5000)/FB Inputs/C{0..8 step 2} Z-Field <-> Data Pointer/HallSensorFieldsXYZ[{32..44 step 3}]  (5 links)
//     Term 7 (APS4322-7000)/Term 8 (APS4322-5000)/FB Inputs/D{1..9 step 2} X-Field <-> Data Pointer/HallSensorFieldsXYZ[{45..57 step 3}]  (5 links)
//     Term 7 (APS4322-7000)/Term 8 (APS4322-5000)/FB Inputs/D{1..9 step 2} Y-Field <-> Data Pointer/HallSensorFieldsXYZ[{46..58 step 3}]  (5 links)
//     Term 7 (APS4322-7000)/Term 8 (APS4322-5000)/FB Inputs/D{1..9 step 2} Z-Field <-> Data Pointer/HallSensorFieldsXYZ[{47..59 step 3}]  (5 links)
//     Term 7 (APS4322-7000)/Term 8 (APS4322-5000)/FB Inputs/E{0..8 step 2} X-Field <-> Data Pointer/HallSensorFieldsXYZ[{60..72 step 3}]  (5 links)
//     Term 7 (APS4322-7000)/Term 8 (APS4322-5000)/FB Inputs/E{0..8 step 2} Y-Field <-> Data Pointer/HallSensorFieldsXYZ[{61..73 step 3}]  (5 links)
//     Term 7 (APS4322-7000)/Term 8 (APS4322-5000)/FB Inputs/E{0..8 step 2} Z-Field <-> Data Pointer/HallSensorFieldsXYZ[{62..74 step 3}]  (5 links)
//     Term 7 (APS4322-7000)/Term 8 (APS4322-5000)/FB Inputs/F{1..9 step 2} X-Field <-> Data Pointer/HallSensorFieldsXYZ[{75..87 step 3}]  (5 links)
//     Term 7 (APS4322-7000)/Term 8 (APS4322-5000)/FB Inputs/F{1..9 step 2} Y-Field <-> Data Pointer/HallSensorFieldsXYZ[{76..88 step 3}]  (5 links)
//     Term 7 (APS4322-7000)/Term 8 (APS4322-5000)/FB Inputs/F{1..9 step 2} Z-Field <-> Data Pointer/HallSensorFieldsXYZ[{77..89 step 3}]  (5 links)
//     Term 7 (APS4322-7000)/Term 8 (APS4322-5000)/FB Inputs/G{0..8 step 2} X-Field <-> Data Pointer/HallSensorFieldsXYZ[{90..102 step 3}]  (5 links)
//     Term 7 (APS4322-7000)/Term 8 (APS4322-5000)/FB Inputs/G{0..8 step 2} Y-Field <-> Data Pointer/HallSensorFieldsXYZ[{91..103 step 3}]  (5 links)
//     Term 7 (APS4322-7000)/Term 8 (APS4322-5000)/FB Inputs/G{0..8 step 2} Z-Field <-> Data Pointer/HallSensorFieldsXYZ[{92..104 step 3}]  (5 links)
//     Term 7 (APS4322-7000)/Term 8 (APS4322-5000)/FB Inputs/H{1..9 step 2} X-Field <-> Data Pointer/HallSensorFieldsXYZ[{105..117 step 3}]  (5 links)
//     Term 7 (APS4322-7000)/Term 8 (APS4322-5000)/FB Inputs/H{1..9 step 2} Y-Field <-> Data Pointer/HallSensorFieldsXYZ[{106..118 step 3}]  (5 links)
//     Term 7 (APS4322-7000)/Term 8 (APS4322-5000)/FB Inputs/H{1..9 step 2} Z-Field <-> Data Pointer/HallSensorFieldsXYZ[{107..119 step 3}]  (5 links)
//     Term 7 (APS4322-7000)/Term 8 (APS4322-5000)/FB Inputs/I{0..8 step 2} X-Field <-> Data Pointer/HallSensorFieldsXYZ[{120..132 step 3}]  (5 links)
//     Term 7 (APS4322-7000)/Term 8 (APS4322-5000)/FB Inputs/I{0..8 step 2} Y-Field <-> Data Pointer/HallSensorFieldsXYZ[{121..133 step 3}]  (5 links)
//     Term 7 (APS4322-7000)/Term 8 (APS4322-5000)/FB Inputs/I{0..8 step 2} Z-Field <-> Data Pointer/HallSensorFieldsXYZ[{122..134 step 3}]  (5 links)
//     Term 7 (APS4322-7000)/Term 8 (APS4322-5000)/FB Inputs/J{1..9 step 2} X-Field <-> Data Pointer/HallSensorFieldsXYZ[{135..147 step 3}]  (5 links)
//     Term 7 (APS4322-7000)/Term 8 (APS4322-5000)/FB Inputs/J{1..9 step 2} Y-Field <-> Data Pointer/HallSensorFieldsXYZ[{136..148 step 3}]  (5 links)
//     Term 7 (APS4322-7000)/Term 8 (APS4322-5000)/FB Inputs/J{1..9 step 2} Z-Field <-> Data Pointer/HallSensorFieldsXYZ[{137..149 step 3}]  (5 links)
//     Term 7 (APS4322-7000)/Term 8 (APS4322-5000)/FB Inputs/Status <-> Data Pointer/FeedbackStatus
//   XPlanar MC Project/Axes/Mover4220_1 <-> TcCOM Objects/XPlanar/Mover4220_1
//     IoToMc/STD <-> OutputsToNC3/HWToNC3
//     McToIo/STD <-> InputsFromNC3/NC3ToHW
//   XPlanar MC Project/Axes/Mover4220_2 <-> TcCOM Objects/XPlanar/Mover4220_2
//     McToIo/STD <-> InputsFromNC3/NC3ToHW
//   XPlanar MC Project/Axes/Mover4220_3 <-> TcCOM Objects/XPlanar/Mover4220_3
//     IoToMc/STD <-> OutputsToNC3/HWToNC3
//   Sim2Real/Sim2Real Instance <-> XPlanar MC Project/Axes/Mover4220_1
//     PlcTask Inputs/GVL.aMovers[1].MCTOPLC/ACT <-> McToPlc/ACT
//     PlcTask Inputs/GVL.aMovers[1].MCTOPLC/COORDMODE <-> McToPlc/COORDMODE
//     PlcTask Inputs/GVL.aMovers[1].MCTOPLC/SET <-> McToPlc/SET
//     PlcTask Inputs/GVL.aMovers[1].MCTOPLC/SETONTRACK <-> McToPlc/SETONTRACK
//     PlcTask Inputs/GVL.aMovers[1].MCTOPLC/STD <-> McToPlc/STD
//     PlcTask Outputs/GVL.aMovers[1].PLCTOMC/STD <-> PlcToMc/STD
//   Sim2Real/Sim2Real Instance <-> XPlanar MC Project/Axes/Mover4220_2
//     PlcTask Inputs/GVL.aMovers[2].MCTOPLC/ACT <-> McToPlc/ACT
//     PlcTask Inputs/GVL.aMovers[2].MCTOPLC/COORDMODE <-> McToPlc/COORDMODE
//     PlcTask Inputs/GVL.aMovers[2].MCTOPLC/SET <-> McToPlc/SET
//     PlcTask Inputs/GVL.aMovers[2].MCTOPLC/SETONTRACK <-> McToPlc/SETONTRACK
//     PlcTask Inputs/GVL.aMovers[2].MCTOPLC/STD <-> McToPlc/STD
//     PlcTask Outputs/GVL.aMovers[2].PLCTOMC/STD <-> PlcToMc/STD
//   Sim2Real/Sim2Real Instance <-> XPlanar MC Project/Axes/Mover4220_3
//     PlcTask Inputs/GVL.aMovers[3].MCTOPLC/ACT <-> McToPlc/ACT
//     PlcTask Inputs/GVL.aMovers[3].MCTOPLC/COORDMODE <-> McToPlc/COORDMODE
//     PlcTask Inputs/GVL.aMovers[3].MCTOPLC/SET <-> McToPlc/SET
//     PlcTask Inputs/GVL.aMovers[3].MCTOPLC/SETONTRACK <-> McToPlc/SETONTRACK
//     PlcTask Inputs/GVL.aMovers[3].MCTOPLC/STD <-> McToPlc/STD
//     PlcTask Outputs/GVL.aMovers[3].PLCTOMC/STD <-> PlcToMc/STD
//   TcCOM Objects/XPlanar/Mover4220_2 <-> XPlanar MC Project/Axes/Mover4220_2
//     OutputsToNC3/HWToNC3 <-> IoToMc/STD
//   TcCOM Objects/XPlanar/Mover4220_3 <-> XPlanar MC Project/Axes/Mover4220_3
//     InputsFromNC3/NC3ToHW <-> McToIo/STD

CONFIGURATION Sim2Real
    RESOURCE PLC ON TwinCAT3
        TASK PlcTask(INTERVAL := T#1ms, PRIORITY := 8);
        PROGRAM MAIN WITH PlcTask : MAIN;
    END_RESOURCE
END_CONFIGURATION

// ---- GVLs/GVL.TcGVL
{attribute 'qualified_only'}
VAR_GLOBAL
	// XPlanar
	aMovers 						: ARRAY[1..nNumMovers] OF MC_PlanarMover;
	aMoverPos 						: ARRAY[1..GVL.nNumMovers] OF MoverVector;
	aMoverVelosDesired				: ARRAY[1..GVL.nNumMovers] OF MoverVector;
	aMoverVelosCurrent				: ARRAY[1..GVL.nNumMovers] OF MoverVector;
	aMoverAccs 						: ARRAY[1..GVL.nNumMovers] OF MoverVector;
	bAllMoversEnabled 				: BOOL;
	bExtSetpointGenActive 			: BOOL := FALSE;
	bExtSetpointGenStart			: BOOL := FALSE;
	fMoverZPos						: LREAL;
	                        		
	// Planning             		
	aSimState						: ARRAY[1..GVL.nNumMovers*6] OF REAL;
	aMoverGoalsXSim 				: ARRAY[1..GVL.nNumMovers] OF REAL;
	aMoverGoalsYSim 				: ARRAY[1..GVL.nNumMovers] OF REAL;
	aMoverAccsDebug					: ARRAY[1..GVL.nNumMovers] OF MoverVector;
	aCntGoals						: ARRAY[1..GVL.nNumMovers] OF UDINT;
	                        		
	// RNG                  		
	fbDrand 						: DRAND;
	                        		
	// Benchmarks           		
	nNumGoalsGenerated 				: DINT := 0;
	aNumGoalsReached 				: ARRAY[1..GVL.nNumMovers] OF DINT := [GVL.nNumMovers(0)];
	aNumCycles1KGoalsReachedSingle	: ARRAY[1..GVL.nNumMovers] OF DINT := [GVL.nNumMovers(0)];
	nNumCycles3KGoalsReachedAll 	: DINT := 0;
	nNumGoalsToGenerate				: DINT := 15000; // success rate
	nNumGoalsToReachPerMover		: DINT := 1000; // makespan
	nNumGoalsToReachAllMovers		: DINT := 3000; // throughput
	nCounterTimeout			  		: DINT := 0;
	nNumCyclesTimeout				: DINT := 120 * 50;
	nNumTimeouts					: DINT := 0;
	nNumGoalsMoverEnd				: DINT := 0;
	aLastGoalMeasured				: ARRAY[1..GVL.nNumMovers] OF BOOL := [GVL.nNumMovers(FALSE)];
 	
	// Paths                	
	fbGetWindowsUser				: FB_GetWindowsUser;
	sWindowsUser					: STRING(255);
	sRelProjectPath					: STRING(255) := '\Documents\TcXaeShell\TC_MagBotSim_Sim2Real\';  // relative to C:\Users\%user% 
	sProjectPath					: STRING(255);
	sVisPath						: STRING(255);
	sFnVisExe						: STRING(255);	
	                        	
	// ML model (policy)    	
	fbMLPredict 					: FB_MllPrediction;	
	nMaxConcurrency 				: UINT := 1;
	sModelFileName					: STRING(255) := 'models\xml\PlanningPolicy_NumMovers_3_LearnJerk_False_NumCycles_120_Vmax_2.0_Amax_10.0.xml';
	sModelFile 						: STRING(255);  // full path to mode file
	nInputDim						: UDINT;
	nOutputDim						: UDINT;
	bPreferredIODataType 			: BOOL;
	bSupportedIODataType 			: BOOL;
	eDtype 							: ETcMllDataType := ETcMllDataType.E_MLLDT_FP32_REAL;
	                        		
	// Visu                 		
	bBeamer 						: BOOL := TRUE;
	bVisualizeGoals		 			: BOOL := TRUE;
END_VAR

VAR_GLOBAL CONSTANT
	// XPlanar
	nNumMovers 			: UINT := 3; // number of movers/agents
	fMaxVelo 			: LREAL := 2000; // [mm/s]
	fMaxAcc 			: LREAL := 10000; // [mm/s^2]
	
	// Policy
	nPolicyInputDim		: UDINT := 3*2*GVL.nNumMovers;
	nPolicyOutputDim 	: UDINT := 2*GVL.nNumMovers;
	fActionSpaceLow		: REAL := -10.0; // [m/s^2]
	fActionSpaceHigh	: REAL := 10.0; // [m/s^2]
	
	
	// Goals and movers
	fMoverSizeSim 		: REAL := 0.113; // [m]
	fThresholdPosSim    : REAL := 0.1; // [m]
	fEpsilon 			: REAL 	:= 0.043; // [m]
	aNumTilesXY 		: ARRAY[1..2] OF UINT := [4,3];
	aSizeFieldSim 		: ARRAY[1..2] OF REAL := [TO_REAL(GVL.aNumTilesXY[1])*0.24, TO_REAL(GVL.aNumTilesXY[2])*0.24]; // [m]
	aMinPosSim 			: ARRAY[1..2] OF REAL := [0.09,0.09];//[GVL.fMoverSizeSim + GVL.fEpsilon, GVL.fMoverSizeSim + GVL.fEpsilon]; // [m], [min_x, min_y]
	aMaxPosSim 			: ARRAY[1..2] OF REAL := [0.81,0.57];//[GVL.aSizeFieldSim[1] - GVL.fMoverSizeSim - GVL.fEpsilon,  GVL.aSizeFieldSim[2] - GVL.fMoverSizeSim - GVL.fEpsilon]; // [m], [max_x, max_y]
	
	// RNG
	nSeed 				: INT := 22;
	
	// Planning
	fDTPrio 			: REAL := 0.001; // s
	nNumCycles			: UDINT := 120;
END_VAR

// ---- POUs/MAIN.TcPOU
PROGRAM MAIN
VAR
	bStart 		: BOOL;
	bStop 		: BOOL;
	bError 		: BOOL;
	nState 		: UDINT := 0; // state machine
	nIdxMover 	: UDINT := 1; // mover index
	
	nIdxPolicyOutput : UDINT;
	
	bAllMoversBusy	: BOOL;
	bAllMoversDone	: BOOL;
	nCycleCounter	: UDINT := 1;
	
	aPolicyOutputScaled	: ARRAY[1..GVL.nPolicyOutputDim] OF REAL;
	aPolicyOutputUnscaled	: ARRAY[1..GVL.nPolicyOutputDim] OF REAL;
	
	nSumMoversEnabled 	: UDINT := 0;
	nSumMoversDone		: UDINT := 0;
	
	aMCPlanarFeedback	: ARRAY[1..GVL.nNumMovers] OF MC_PlanarFeedback;
	stOptionsESG 		: ST_ExternalSetpointGenerationOptions;
	stMoveCOptions		: ST_MoveCOptions;
	iDynConstraint		: IPlcDynamicConstraint;
	
	fbStartProcess 		: NT_StartProcess;
	fbTimer				: TON;
	tTime				: TIME := T#0D0H0M10S0MS;
	
	fbXPlanarEnvironment		: FB_TcIoXPlanarEnvironment;
	bInitXPlanarEnv				: BOOL := TRUE;
	MoverCommunicationStatus	: CoordinatedMoverCommStatus;
	
	fXPosMover  : REAL;
	fYPosMover	: REAL;
	
	nSumGoalsReachedAllMovers 			: DINT := 0;
	bBenchmarkReachedPerMoverFinished 	: BOOL := FALSE;
	bBenchmarkReachedAllFinished 		: BOOL := FALSE;
	bBenchmarkSuccessRateFinished 		: BOOL := FALSE;
	
	
	nCounterNoGoalReached			: UDINT := 0;
END_VAR

CASE nState OF
	0:  // build all paths
		GVL.fbGetWindowsUser();
		IF GVL.fbGetWindowsUser.bDone THEN
			GVL.sWindowsUser := GVL.fbGetWindowsUser.sUser;
			GVL.sProjectPath := concat(concat('C:\Users\', GVL.sWindowsUser), GVL.sRelProjectPath);
			GVL.sVisPath := concat(GVL.sProjectPath,'visualization');
			GVL.sFnVisExe := concat(GVL.sVisPath, '\dist\demo.exe');			
			GVL.sModelFile := concat(GVL.sProjectPath, GVL.sModelFileName);
			nState := 1;
		END_IF

	1:	// wait for start
		IF bStart AND NOT bStop AND NOT bError THEN
			bStart := FALSE;
			bStop := FALSE;
			bAllMoversBusy := FALSE;
			bAllMoversDone := FALSE;
			GVL.bVisualizeGoals := TRUE;
			GVL.bExtSetpointGenActive := FALSE;
			GVL.bAllMoversEnabled := FALSE;
			GVL.fbDrand(Seed := GVL.nSeed);
			fbTimer.IN := FALSE; // reset timer
			
			FOR nIdxMover := 1 TO GVL.nNumMovers DO
				GVL.aNumGoalsReached[nIdxMover] := 0;
				GVL.aNumCycles1KGoalsReachedSingle[nIdxMover] := 0;
			END_FOR
			GVL.nNumCycles3KGoalsReachedAll := 0;
			nSumGoalsReachedAllMovers := 0;
			bBenchmarkReachedPerMoverFinished := FALSE;
			bBenchmarkReachedAllFinished := FALSE;
			bBenchmarkSuccessRateFinished := FALSE;
			GVL.nNumTimeouts := 0;
			
			nState := 10;
		END_IF
		
	10: // init env
		IF bInitXPlanarEnv THEN
			IF fbXPlanarEnvironment.Init(TRUE) THEN
				fbXPlanarEnvironment.Init(FALSE);
				bInitXPlanarEnv := FALSE;
				nState := nState + 1;
			END_IF
		ELSE
			nState := nState + 1;
		END_IF
	
	11:// mover communication
		IF fbXPlanarEnvironment.XpuTcIo(1).SetCoordMoverCommunicationCmd(CoordinatedMoverCommCommand.IdentifyAndAssignPossible) THEN
			nState := nState + 1;
		END_IF
		
	12: // check mover communication
		MoverCommunicationStatus := fbXPlanarEnvironment.XpuTcIo(1).GetCoordMoverCommStatus();
		IF MoverCommunicationStatus = CoordinatedMoverCommStatus.CommunicationSuccessful THEN
			nState := 20;
		END_IF

	20:	// load policy
		GVL.fbMLPredict.stPredictionParameter.MaxConcurrency := GVL.nMaxConcurrency;
		GVL.fbMLPredict.stPredictionParameter.MlModelFilepath := GVL.sModelFile;				
		IF GVL.fbMLPredict.Configure() THEN
			// check input and output dimensions and data type
			bError := GVL.fbMLPredict.GetInputDim(GVL.nInputDim);
			bError := GVL.fbMLPredict.GetOutputDim(GVL.nOutputDim);
			bError := GVL.fbMLPredict.CheckPreferredIODataTypes(ETcMllDataType.E_MLLDT_FP32_REAL,ETcMllDataType.E_MLLDT_FP32_REAL,GVL.bPreferredIODataType);
			bError := GVL.fbMlPredict.CheckSupportedIODataTypes(ETcMllDataType.E_MLLDT_FP32_REAL,ETcMllDataType.E_MLLDT_FP32_REAL,GVL.bSupportedIODataType);
		
			IF GVL.bPreferredIODataType OR GVL.bSupportedIODataType THEN
				GVL.eDtype := ETcMllDataType.E_MLLDT_FP32_REAL;
			END_IF
			
			IF bError OR GVL.fbMLPredict.bError OR GVL.nInputDim <> GVL.nPolicyInputDim OR GVL.nOutputDim <> GVL.nPolicyOutputDim THEN
				nState := 999;
			ELSE
				nState := 30;
			END_IF
		END_IF
 
		
	30:
		fbStartProcess.START := TRUE;
		IF fbStartProcess.BUSY THEN
			fbTimer.IN := TRUE;
			nState := nState + 1;
		END_IF
		
	31:
		fbStartProcess.START := FALSE;
		IF NOT fbStartProcess.BUSY AND fbTimer.Q THEN
			nState := 40;
		END_IF

	40: // enable all movers
		FOR nIdxMover := 1 TO GVL.nNumMovers DO
			GVL.aMovers[nIdxMover].Enable(0);
		END_FOR
		nState := nState + 1;
		
	41:	// wait until all movers are enabled
		nSumMoversEnabled := 0;
		FOR nIdxMover := 1 TO GVL.nNumMovers DO
			IF GVL.aMovers[nIdxMover].MCTOPLC.STD.State = MC_PLANAR_STATE.Enabled THEN
				nSumMoversEnabled := nSumMoversEnabled + 1;
			END_IF
		END_FOR
		IF nSumMoversEnabled = GVL.nNumMovers THEN
			GVL.bAllMoversEnabled := TRUE;
			nState := nState + 1;
		END_IF
		
	42: // move C
		FOR nIdxMover := 1 TO GVL.nNumMovers DO
			GVL.aMovers[nIdxMover].MoveC(commandFeedback := aMCPlanarFeedback[nIdxMover], targetPosition := 0.0, constraint := 0, options := 0);
		END_FOR
		nState := nState + 1;
		
	43:
		nSumMoversDone := 0;
		FOR nIdxMover := 1 TO GVL.nNumMovers DO
			IF aMCPlanarFeedback[nIdxMover].Done THEN
				nSumMoversDone := nSumMoversDone + 1;
			END_IF
		END_FOR
		IF nSumMoversDone = GVL.nNumMovers THEN
			nState := 50;
		END_IF
	
	50: // sample first goals
		FOR nIdxMover := 1 TO GVL.nNumMovers DO
			M_SampleGoal(nIdxMover := nIdxMover);
			GVL.nNumGoalsGenerated := GVL.nNumGoalsGenerated + 1;
		END_FOR
		nState := 70;
		
	70:	// prepare desired positions, velocities and accelerations before starting external setpoint generation
		GVL.fMoverZPos := GVL.aMovers[1].MCTOPLC.ACT.ActPos.z;
		FOR nIdxMover := 1 TO GVL.nNumMovers DO
			// start position = current position of the mover
			GVL.aMoverPos[nIdxMover] := GVL.aMovers[nIdxMover].MCTOPLC.ACT.ActPos;
			// start velocities 
			GVL.aMoverVelosDesired[nIdxMover].x := 0.0;
			GVL.aMoverVelosDesired[nIdxMover].y := 0.0;
			GVL.aMoverVelosDesired[nIdxMover].z := 0.0;
			GVL.aMoverVelosDesired[nIdxMover].a := 0.0;
			GVL.aMoverVelosDesired[nIdxMover].b := 0.0;
			GVL.aMoverVelosDesired[nIdxMover].c := 0.0;
			
			GVL.aMoverVelosCurrent[nIdxMover].x := 0.0;
			GVL.aMoverVelosCurrent[nIdxMover].y := 0.0;
			GVL.aMoverVelosCurrent[nIdxMover].z := 0.0;
			GVL.aMoverVelosCurrent[nIdxMover].a := 0.0;
			GVL.aMoverVelosCurrent[nIdxMover].b := 0.0;
			GVL.aMoverVelosCurrent[nIdxMover].c := 0.0;
			// start accelerations 
			GVL.aMoverAccs[nIdxMover].x := 0.0;
			GVL.aMoverAccs[nIdxMover].y := 0.0;
			GVL.aMoverAccs[nIdxMover].z := 0.0;
			GVL.aMoverAccs[nIdxMover].a := 0.0;
			GVL.aMoverAccs[nIdxMover].b := 0.0;
			GVL.aMoverAccs[nIdxMover].c := 0.0;
		END_FOR
		nState := nState + 1;
		
	71: // start external setpoint generation for each mover
		stOptionsESG.mode := MC_EXTERNAL_SET_POSITION_MODE.Absolute;
		FOR nIdxMover := 1 TO GVL.nNumMovers DO
			GVL.aMovers[nIdxMover].StartExternalSetpointGeneration(aMCPlanarFeedback[nIdxMover],stOptionsESG);
		END_FOR
		nState := nState + 1;
		
	72: // wait until external setpoint generation is active
		nSumMoversDone := 0;
		FOR nIdxMover := 1 TO GVL.nNumMovers DO
			IF aMCPlanarFeedback[nIdxMover].Done THEN
				nSumMoversDone := nSumMoversDone + 1;
			END_IF
		END_FOR
		IF nSumMoversDone = GVL.nNumMovers THEN
			GVL.bExtSetpointGenActive := TRUE;
			GVL.bExtSetpointGenStart := TRUE;
			nCycleCounter := 0;
			nState := 80;
		END_IF
		
	80: // planning - stop or set new accelerations
		IF bStop OR bError OR (bBenchmarkReachedPerMoverFinished AND bBenchmarkReachedAllFinished AND bBenchmarkSuccessRateFinished) THEN
			// stop external setpoint generation
			nState := 200;
		ELSIF nCycleCounter = 0 OR nCycleCounter > GVL.nNumCycles THEN
			GVL.fbMLPredict.Predict(
					pDataInp := ADR(GVL.aSimState), 
					nDataInpDim := GVL.nPolicyInputDim, 
					fmtDataInpType:= GVL.eDtype, 
					pDataOut:= ADR(aPolicyOutputScaled), 
					nDataOutDim:= GVL.nPolicyOutputDim, 
					fmtDataOutType:= GVL.eDtype, 
					nEngineId:= 0, // only one engine available in this model
					nConcurrencyId:=0);
					
			FOR nIdxPolicyOutput := 1 TO GVL.nPolicyOutputDim DO
				// undo action scaling
				aPolicyOutputUnscaled[nIdxPolicyOutput] := GVL.fActionSpaceLow + (0.5 * (aPolicyOutputScaled[nIdxPolicyOutput] + 1.0) * (GVL.fActionSpaceHigh - GVL.fActionSpaceLow));
			END_FOR
			FOR nIdxMover := 1 TO GVL.nNumMovers DO
				GVL.aMoverAccs[nIdxMover].x := aPolicyOutputUnscaled[(nIdxMover - 1) * 2 + 1] * 1000.0;
				GVL.aMoverAccs[nIdxMover].y := aPolicyOutputUnscaled[(nIdxMover - 1) * 2 + 2] * 1000.0;
			END_FOR
			nCycleCounter := 1;
		ELSE
			nCycleCounter := nCycleCounter + 1;
		END_IF
		
		// benchmarks
		bBenchmarkReachedPerMoverFinished := TRUE;
		nSumGoalsReachedAllMovers := 0;
		// makespan
		FOR nIdxMover := 1 TO GVL.nNumMovers DO
			nSumGoalsReachedAllMovers := nSumGoalsReachedAllMovers + GVL.aNumGoalsReached[nIdxMover];
			IF GVL.aNumGoalsReached[nIdxMover] < GVL.nNumGoalsToReachPerMover THEN
				GVL.aNumCycles1KGoalsReachedSingle[nIdxMover] := GVL.aNumCycles1KGoalsReachedSingle[nIdxMover] + 1;
				bBenchmarkReachedPerMoverFinished := bBenchmarkReachedPerMoverFinished AND (GVL.aNumGoalsReached[nIdxMover] >= GVL.nNumGoalsToReachPerMover);
			END_IF
		END_FOR
		// throughput
		IF nSumGoalsReachedAllMovers < GVL.nNumGoalsToReachAllMovers THEN
			bBenchmarkReachedAllFinished := FALSE;
			GVL.nNumCycles3KGoalsReachedAll := GVL.nNumCycles3KGoalsReachedAll + 1;
		ELSE
			bBenchmarkReachedAllFinished := TRUE;
		END_IF
		
	200:// stop external setpoint generation, all movers will reduce their velocity to 0 (automatically)
		GVL.bExtSetpointGenStart := FALSE;
		FOR nIdxMover := 1 TO GVL.nNumMovers DO
			GVL.aMovers[nIdxMover].StopExternalSetpointGeneration(aMCPlanarFeedback[nIdxMover]);
		END_FOR
		nState := nState + 1;
		
	201:// wait until external setpoint generation is stopped
		nSumMoversDone := 0;
		FOR nIdxMover := 1 TO GVL.nNumMovers DO
			IF aMCPlanarFeedback[nIdxMover].Done THEN
				nSumMoversDone := nSumMoversDone + 1;
			END_IF
		END_FOR
		IF nSumMoversDone = GVL.nNumMovers THEN
			GVL.bExtSetpointGenActive := FALSE;
			nState := nState + 1;
		END_IF	
		
	202:// disable all movers
		FOR nIdxMover := 1 TO GVL.nNumMovers DO
			GVL.aMovers[nIdxMover].Disable(aMCPlanarFeedback[nIdxMover]);
		END_FOR
		nState := nState + 1;
		
	203:// wait until all movers are disabled
		nSumMoversDone := 0;
		FOR nIdxMover := 1 TO GVL.nNumMovers DO
			IF NOT aMCPlanarFeedback[nIdxMover].Done THEN
				nSumMoversDone := nSumMoversDone + 1;
			END_IF
		END_FOR
		IF nSumMoversDone = GVL.nNumMovers THEN
			GVL.bAllMoversEnabled := FALSE;
			nState := 1;
		END_IF
	
	999: // error state
		GVL.bExtSetpointGenStart := FALSE;
		bError := TRUE;
		IF GVL.bExtSetpointGenActive THEN
			// stop external setpoint generation
			nState := 200; 
		END_IF
		
END_CASE

IF nState > 1 THEN
	nCounterNoGoalReached := 0;
	FOR nIdxMover := 1 TO GVL.nNumMovers DO
		IF GVL.bExtSetpointGenActive AND GVL.bExtSetpointGenStart THEN
			// velocity
			GVL.aMoverVelosCurrent[nIdxMover].x := GVL.aMoverVelosDesired[nIdxMover].x + (GVL.fDTPrio * GVL.aMoverAccs[nIdxMover].x);
			GVL.aMoverVelosCurrent[nIdxMover].y := GVL.aMoverVelosDesired[nIdxMover].y + (GVL.fDTPrio * GVL.aMoverAccs[nIdxMover].y);
			GVL.aMoverVelosDesired[nIdxMover].x := GVL.aMoverVelosCurrent[nIdxMover].x;
			GVL.aMoverVelosDesired[nIdxMover].y := GVL.aMoverVelosCurrent[nIdxMover].y;
			IF F_EnsureMaxVelo(fNextVeloX := GVL.aMoverVelosDesired[nIdxMover].x, fNextVeloY := GVL.aMoverVelosDesired[nIdxMover].y) THEN
				GVL.aMoverAccs[nIdxMover].x := (GVL.aMoverVelosCurrent[nIdxMover].x - GVL.aMoverVelosDesired[nIdxMover].x)/GVL.fDTPrio;
				GVL.aMoverAccs[nIdxMover].y := (GVL.aMoverVelosCurrent[nIdxMover].y - GVL.aMoverVelosDesired[nIdxMover].y)/GVL.fDTPrio;
			END_IF
			GVL.aMoverVelosDesired[nIdxMover].z := GVL.fMoverZPos - GVL.aMoverPos[nIdxMover].z;	
		
			// position
			GVL.aMoverPos[nIdxMover].x := GVL.aMoverPos[nIdxMover].x + (GVL.fDTPrio * GVL.aMoverVelosDesired[nIdxMover].x);
			GVL.aMoverPos[nIdxMover].y := GVL.aMoverPos[nIdxMover].y + (GVL.fDTPrio * GVL.aMoverVelosDesired[nIdxMover].y);
			GVL.aMoverPos[nIdxMover].z := GVL.fMoverZPos;
			
			// set new setpoint
			GVL.aMovers[nIdxMover].SetExternalSetpoint(GVL.aMoverPos[nIdxMover],GVL.aMoverVelosDesired[nIdxMover],GVL.aMoverAccs[nIdxMover]);
		END_IF
		// update mover state and command feedback
		GVL.aMovers[nIdxMover].Update();
		aMCPlanarFeedback[nIdxMover].Update();
		// update mover sim state
		M_GetSimState(aSimState => GVL.aSimState);
		// check errors
		IF (GVL.aMovers[nIdxMover].Error OR aMCPlanarFeedback[nIdxMover].Error) AND nState < 200 AND nState <> 1 THEN
			nState := 999;
		END_IF
		// check goal reached
		IF M_CheckGoalReached(nIdxMover := nIdxMover) THEN
			// if goal is reached: sample new goal, else: use old goal
			IF GVL.nNumGoalsGenerated < GVL.nNumGoalsToGenerate THEN
				GVL.aNumGoalsReached[nIdxMover] := GVL.aNumGoalsReached[nIdxMover] + 1;
				M_SampleGoal(nIdxMover := nIdxMover);
				GVL.nNumGoalsGenerated := GVL.nNumGoalsGenerated + 1;
				IF GVL.nNumGoalsGenerated = GVL.nNumGoalsToGenerate THEN
					GVL.nCounterTimeout := -1;
					
					nSumGoalsReachedAllMovers := 0;
					// makespan
					FOR nIdxMover := 1 TO GVL.nNumMovers DO
						nSumGoalsReachedAllMovers := nSumGoalsReachedAllMovers + GVL.aNumGoalsReached[nIdxMover];
					END_FOR
					GVL.nNumGoalsMoverEnd := nSumGoalsReachedAllMovers;
					EXIT;
				END_IF
			ELSIF NOT GVL.aLastGoalMeasured[nIdxMover] THEN
				GVL.aNumGoalsReached[nIdxMover] := GVL.aNumGoalsReached[nIdxMover] + 1;
				GVL.aLastGoalMeasured[nIdxMover] := TRUE;
			END_IF
		ELSE
			nCounterNoGoalReached := nCounterNoGoalReached + 1;
		END_IF
	END_FOR
	IF nState = 80 THEN
		// check whether timeout counter must be increased or resetted
		IF nCounterNoGoalReached = GVL.nNumMovers OR GVL.nNumGoalsGenerated >= GVL.nNumGoalsToGenerate THEN
			GVL.nCounterTimeout := GVL.nCounterTimeout + 1;
		ELSE
			GVL.nCounterTimeout := 0;
		END_IF
		// if timeout, sample new goals for all movers
		IF GVL.nCounterTimeout = GVL.nNumCyclesTimeout THEN
			GVL.nNumTimeouts := GVL.nNumTimeouts + 1;
			IF GVL.nNumGoalsGenerated >= GVL.nNumGoalsToGenerate THEN
				bBenchmarkSuccessRateFinished := TRUE;
			END_IF
			IF NOT bBenchmarkSuccessRateFinished OR NOT bBenchmarkReachedPerMoverFinished OR NOT bBenchmarkReachedAllFinished THEN
				FOR nIdxMover := 1 TO GVL.nNumMovers DO
					M_SampleGoal(nIdxMover := nIdxMover);
					GVL.nNumGoalsGenerated := GVL.nNumGoalsGenerated + 1;
				END_FOR
				GVL.nCounterTimeout := 0;
				nCycleCounter := 0;	
			END_IF
		ELSIF GVL.nNumGoalsGenerated >= GVL.nNumGoalsToGenerate AND nSumGoalsReachedAllMovers = (GVL.nNumGoalsMoverEnd + GVL.nNumMovers) THEN
			bBenchmarkSuccessRateFinished := TRUE;
		END_IF
	END_IF
		
	// visualization
	fbStartProcess(PATHSTR := GVL.sFnVisExe);
	IF fbStartProcess.ERR THEN
		nState := 999;
	END_IF
	fbTimer(PT := tTime);
END_IF

METHOD M_CheckGoalReached : BOOL
VAR_INPUT
	nIdxMover : UDINT; // mover index
END_VAR
	
VAR
	fDiffXSim : REAL;
	fDiffYSim : REAL;
END_VAR
fDiffXSim := GVL.aMoverGoalsXSim[nIdxMover] - (TO_REAL(GVL.aMovers[nIdxMover].MCTOPLC.SET.SetPos.x) * 0.001); // [m]
fDiffYSim := GVL.aMoverGoalsYSim[nIdxMover] - (TO_REAL(GVL.aMovers[nIdxMover].MCTOPLC.SET.SetPos.y) * 0.001); // [m]

IF F_2Norm(fA := fDiffXSim, fB := fDiffYSim) < GVL.fThresholdPosSim THEN
	M_CheckGoalReached := TRUE;
ELSE
	M_CheckGoalReached := FALSE;
END_IF
END_METHOD

METHOD M_GetSimState :  BOOL
VAR
	nIdxMover	: UDINT;
END_VAR

VAR_OUTPUT
	aSimState : ARRAY[1..GVL.nNumMovers*6] OF REAL;
END_VAR
FOR nIdxMover := 1 TO GVL.nNumMovers DO
	// position ("achieved_goal")
	aSimState[(nIdxMover - 1) * 2 + 1] := TO_REAL(GVL.aMovers[nIdxMover].MCTOPLC.ACT.ActPos.x) * 0.001; // [m]
	aSimState[(nIdxMover - 1) * 2 + 2] := TO_REAL(GVL.aMovers[nIdxMover].MCTOPLC.ACT.ActPos.y) * 0.001; // [m]
	// goal ("desired_goal")
	aSimState[(GVL.nNumMovers*2) + (nIdxMover - 1) * 2 + 1] := GVL.aMoverGoalsXSim[nIdxMover];
	aSimState[(GVL.nNumMovers*2) + (nIdxMover - 1) * 2 + 2] := GVL.aMoverGoalsYSim[nIdxMover];
	// velocity ("observation")
	aSimState[(GVL.nNumMovers*2*2) + (nIdxMover - 1) * 2 + 1] := TO_REAL(GVL.aMovers[nIdxMover].MCTOPLC.ACT.ActVelo.x) * 0.001; // [m/s]
	aSimState[(GVL.nNumMovers*2*2) + (nIdxMover - 1) * 2 + 2] := TO_REAL(GVL.aMovers[nIdxMover].MCTOPLC.ACT.ActVelo.y) * 0.001; // [m/s]
END_FOR
M_GetSimState := TRUE;
END_METHOD

METHOD M_SampleGoal
VAR_INPUT
	nIdxMover 			: UDINT; // mover index
END_VAR
VAR 
	fRandomNumber 		: LREAL;
	fDiffXSim 			: REAL;
	fDiffYSim 			: REAL;
	fMoverGoalXSim 		: REAL;
	fMoverGoalYSim 		: REAL;
	fObstacleGoalXSim 	: REAL;
	fObstacleGoalYSim 	: REAL;
	nIdx				: UDINT;
	nSumDistGoalsValid	: UDINT;
END_VAR
// generate x-position of the goal
GVL.fbDrand(num => fRandomNumber);
fMoverGoalXSim := (GVL.aMaxPosSim[1] - GVL.aMinPosSim[1]) * TO_REAL(fRandomNumber) + GVL.aMinPosSim[1]; // [m]
// generate y-position of the goal
GVL.fbDrand(num => fRandomNumber);
fMoverGoalYSim := (GVL.aMaxPosSim[2] - GVL.aMinPosSim[2]) * TO_REAL(fRandomNumber) + GVL.aMinPosSim[2]; // [m]

GVL.aMoverGoalsXSim[nIdxMover] := fMoverGoalXSim;
GVL.aMoverGoalsYSim[nIdxMover] := fMoverGoalYSim;
END_METHOD

END_PROGRAM

// ---- Functions/F_EnsureMaxVelo.TcPOU
FUNCTION F_EnsureMaxVelo: BOOL
VAR_IN_OUT
	fNextVeloX : LREAL;
	fNextVeloY : LREAL;
END_VAR
VAR
	fNormNextVelo : LREAL;
	fNextVeloUnitLength : LREAL;
END_VAR

fNormNextVelo := TO_LREAL(F_2Norm(fA := TO_REAL(fNextVeloX), fB := TO_REAL(fNextVeloY)));
IF fNormNextVelo > GVL.fMaxVelo THEN
	fNextVeloX := (fNextVeloX/fNormNextVelo) * GVL.fMaxVelo;
	fNextVeloY := (fNextVeloY/fNormNextVelo) * GVL.fMaxVelo;
	F_EnsureMaxVelo := TRUE;
END_IF
F_EnsureMaxVelo := FALSE;

END_FUNCTION

// ---- Functions/F_2Norm.TcPOU
FUNCTION F_2Norm : REAL
VAR_INPUT
	fA : REAL;
	fB : REAL;
END_VAR
VAR
END_VAR

F_2Norm := SQRT(fA*fA + fB*fB);

END_FUNCTION
